LIN {X 0,Y 277.24,Z 414.573,A -85,B 0,C 180,E1 -17493.897,E2 -17493.897} C_VEL
LIN {X 0,Y 277.261,Z 414.56,A -85,B 0,C 180,E1 -17497.471,E2 -17497.471} C_VEL
LIN {X 0,Y 277.204,Z 414.578,A -85,B 0,C 180,E1 -17501.238,E2 -17501.238} C_VEL
LIN {X 0,Y 277.218,Z 414.568,A -85,B 0,C 180,E1 -17505.224,E2 -17505.224} C_VEL
LIN {X 0,Y 277.258,Z 414.57,A -85,B 0,C 180,E1 -17509.504,E2 -17509.504} C_VEL
LIN {X 0,Y 277.287,Z 414.57,A -85,B 0,C 180,E1 -17512.536,E2 -17512.536} C_VEL
LIN {X 0,Y 277.252,Z 414.575,A -85,B 0,C 180,E1 -17516.107,E2 -17516.107} C_VEL
LIN {X 0,Y 277.26,Z 414.568,A -85,B 0,C 180,E1 -17519.541,E2 -17519.541} C_VEL
LIN {X 0,Y 277.358,Z 414.56,A -85,B 0,C 180,E1 -17522.866,E2 -17522.866} C_VEL
LIN {X 0,Y 277.333,Z 414.568,A -85,B 0,C 180,E1 -17527.465,E2 -17527.465} C_VEL
LIN {X 0,Y 278.42,Z 417.605,A -85,B 0,C 180,E1 -17527.717,E2 -17527.717} C_VEL
LIN {X 0,Y 283.895,Z 430.25,A -85,B 0,C 180,E1 -17528.839,E2 -17528.839} C_VEL
LIN {X 0,Y 287.727,Z 441.564,A -85,B 0,C 180,E1 -17530.005,E2 -17530.005} C_VEL
LIN {X 0,Y 288.639,Z 445.273,A -85,B 0,C 180,E1 -17530.418,E2 -17530.418} C_VEL
LIN {X 0,Y 287.704,Z 456.27,A -85,B 0,C 180,E1 -17531.486,E2 -17531.486} C_VEL
LIN {X 0,Y 286.431,Z 467.423,A -85,B 0,C 180,E1 -17532.878,E2 -17532.878} C_VEL
LIN {X 0,Y 284.992,Z 477.37,A -85,B 0,C 180,E1 -17534.423,E2 -17534.423} C_VEL
LIN {X 0,Y 283.633,Z 485.752,A -85,B 0,C 180,E1 -17536.021,E2 -17536.021} C_VEL
LIN {X 0,Y 282.322,Z 493.35,A -85,B 0,C 180,E1 -17537.786,E2 -17537.786} C_VEL
LIN {X 0,Y 280.888,Z 500.786,A -85,B 0,C 180,E1 -17539.915,E2 -17539.915} C_VEL
LIN {X 0,Y 279.945,Z 506.702,A -85,B 0,C 180,E1 -17542.065,E2 -17542.065} C_VEL
LIN {X 0,Y 279.051,Z 511.413,A -85,B 0,C 180,E1 -17544.22,E2 -17544.22} C_VEL
LIN {X 0,Y 278.325,Z 515.036,A -85,B 0,C 180,E1 -17546.382,E2 -17546.382} C_VEL
LIN {X 0,Y 277.829,Z 517.669,A -85,B 0,C 180,E1 -17548.552,E2 -17548.552} C_VEL
LIN {X 0,Y 277.7,Z 519.747,A -85,B 0,C 180,E1 -17551.452,E2 -17551.452} C_VEL
LIN {X 0,Y 277.587,Z 520.2,A -85,B 0,C 180,E1 -17552.904,E2 -17552.904} C_VEL
LIN {X 0,Y 277.489,Z 520.279,A -85,B 0,C 180,E1 -17554.359,E2 -17554.359} C_VEL
LIN {X 0,Y 278.16,Z 519.232,A -85,B 0,C 180,E1 -17557.259,E2 -17557.259} C_VEL
LIN {X 0,Y 278.687,Z 518.077,A -85,B 0,C 180,E1 -17558.704,E2 -17558.704} C_VEL
LIN {X 0,Y 279.649,Z 514.63,A -85,B 0,C 180,E1 -17561.6,E2 -17561.6} C_VEL
LIN {X 0,Y 280.708,Z 510.847,A -85,B 0,C 180,E1 -17563.761,E2 -17563.761} C_VEL
LIN {X 0,Y 281.838,Z 505.952,A -85,B 0,C 180,E1 -17565.922,E2 -17565.922} C_VEL
LIN {X 0,Y 283.221,Z 499.731,A -85,B 0,C 180,E1 -17568.072,E2 -17568.072} C_VEL
LIN {X 0,Y 284.989,Z 491.93,A -85,B 0,C 180,E1 -17570.198,E2 -17570.198} C_VEL
LIN {X 0,Y 286.653,Z 483.93,A -85,B 0,C 180,E1 -17571.957,E2 -17571.957} C_VEL
LIN {X 0,Y 288.379,Z 474.102,A -85,B 0,C 180,E1 -17573.712,E2 -17573.712} C_VEL
LIN {X 0,Y 289.969,Z 462.99,A -85,B 0,C 180,E1 -17575.29,E2 -17575.29} C_VEL
LIN {X 0,Y 291.243,Z 452.011,A -85,B 0,C 180,E1 -17576.52,E2 -17576.52} C_VEL
LIN {X 0,Y 291.418,Z 448.805,A -85,B 0,C 180,E1 -17576.833,E2 -17576.833} C_VEL
LIN {X 0,Y 288.104,Z 438.67,A -85,B 0,C 180,E1 -17578.107,E2 -17578.107} C_VEL
LIN {X 0,Y 283.2,Z 426.913,A -85,B 0,C 180,E1 -17579.437,E2 -17579.437} C_VEL
LIN {X 0,Y 278.243,Z 417.384,A -85,B 0,C 180,E1 -17580.428,E2 -17580.428} C_VEL
LIN {X 0,Y 277.259,Z 414.575,A -85,B 0,C 180,E1 -17580.659,E2 -17580.659} C_VEL
LIN {X 0,Y 277.253,Z 414.579,A -85,B 0,C 180,E1 -17583.896,E2 -17583.896} C_VEL
LIN {X 0,Y 277.27,Z 414.557,A -85,B 0,C 180,E1 -17587.47,E2 -17587.47} C_VEL
LIN {X 0,Y 277.215,Z 414.579,A -85,B 0,C 180,E1 -17591.237,E2 -17591.237} C_VEL
LIN {X 0,Y 277.207,Z 414.574,A -85,B 0,C 180,E1 -17595.227,E2 -17595.227} C_VEL
LIN {X 0,Y 277.228,Z 414.555,A -85,B 0,C 180,E1 -17599.512,E2 -17599.512} C_VEL
LIN {X 0,Y 277.27,Z 414.542,A -85,B 0,C 180,E1 -17602.53,E2 -17602.53} C_VEL
LIN {X 0,Y 277.253,Z 414.573,A -85,B 0,C 180,E1 -17606.104,E2 -17606.104} C_VEL
LIN {X 0,Y 277.267,Z 414.524,A -85,B 0,C 180,E1 -17609.539,E2 -17609.539} C_VEL
LIN {X 0,Y 277.362,Z 414.537,A -85,B 0,C 180,E1 -17612.864,E2 -17612.864} C_VEL
LIN {X 0,Y 277.351,Z 414.616,A -85,B 0,C 180,E1 -17615.497,E2 -17615.497} C_VEL
LIN {X 0,Y 281.258,Z 428.661,A -85,B 0,C 180,E1 -17617.03,E2 -17617.03} C_VEL
LIN {X 0,Y 284.772,Z 441.274,A -85,B 0,C 180,E1 -17618.652,E2 -17618.652} C_VEL
LIN {X 0,Y 285.159,Z 442.879,A -85,B 0,C 180,E1 -17618.872,E2 -17618.872} C_VEL
LIN {X 0,Y 283.769,Z 455.996,A -85,B 0,C 180,E1 -17620.634,E2 -17620.634} C_VEL
LIN {X 0,Y 282.205,Z 468.131,A -85,B 0,C 180,E1 -17622.611,E2 -17622.611} C_VEL
LIN {X 0,Y 280.871,Z 479.118,A -85,B 0,C 180,E1 -17624.767,E2 -17624.767} C_VEL
LIN {X 0,Y 279.838,Z 488.37,A -85,B 0,C 180,E1 -17626.936,E2 -17626.936} C_VEL
LIN {X 0,Y 278.893,Z 497.005,A -85,B 0,C 180,E1 -17629.359,E2 -17629.359} C_VEL
LIN {X 0,Y 278.249,Z 504.77,A -85,B 0,C 180,E1 -17632.014,E2 -17632.014} C_VEL
LIN {X 0,Y 277.657,Z 509.994,A -85,B 0,C 180,E1 -17634.189,E2 -17634.189} C_VEL
LIN {X 0,Y 277.409,Z 514.29,A -85,B 0,C 180,E1 -17636.368,E2 -17636.368} C_VEL
LIN {X 0,Y 277.436,Z 515.059,A -85,B 0,C 180,E1 -17636.807,E2 -17636.807} C_VEL
LIN {X 0,Y 276.857,Z 517.048,A -85,B 0,C 180,E1 -17637.951,E2 -17637.951} C_VEL
LIN {X 0,Y 274.139,Z 520.047,A -85,B 0,C 180,E1 -17639.836,E2 -17639.836} C_VEL
LIN {X 0,Y 271.891,Z 522.007,A -85,B 0,C 180,E1 -17641.391,E2 -17641.391} C_VEL
LIN {X 0,Y 271.052,Z 523.132,A -85,B 0,C 180,E1 -17642.61,E2 -17642.61} C_VEL
LIN {X 0,Y 271.055,Z 523.425,A -85,B 0,C 180,E1 -17643.024,E2 -17643.024} C_VEL
LIN {X 0,Y 271.926,Z 525.003,A -85,B 0,C 180,E1 -17645.934,E2 -17645.934} C_VEL
LIN {X 0,Y 273.318,Z 525.329,A -85,B 0,C 180,E1 -17648.875,E2 -17648.875} C_VEL
LIN {X 0,Y 275.228,Z 524.402,A -85,B 0,C 180,E1 -17651.787,E2 -17651.787} C_VEL
LIN {X 0,Y 277.652,Z 522.226,A -85,B 0,C 180,E1 -17654.662,E2 -17654.662} C_VEL
LIN {X 0,Y 280.567,Z 518.782,A -85,B 0,C 180,E1 -17657.493,E2 -17657.493} C_VEL
LIN {X 0,Y 284.117,Z 513.978,A -85,B 0,C 180,E1 -17660.261,E2 -17660.261} C_VEL
LIN {X 0,Y 288.296,Z 507.671,A -85,B 0,C 180,E1 -17662.957,E2 -17662.957} C_VEL
LIN {X 0,Y 293.036,Z 499.73,A -85,B 0,C 180,E1 -17665.575,E2 -17665.575} C_VEL
LIN {X 0,Y 297.591,Z 491.324,A -85,B 0,C 180,E1 -17667.802,E2 -17667.802} C_VEL
LIN {X 0,Y 302.538,Z 481.329,A -85,B 0,C 180,E1 -17669.929,E2 -17669.929} C_VEL
LIN {X 0,Y 304.146,Z 477.942,A -85,B 0,C 180,E1 -17670.554,E2 -17670.554} C_VEL
LIN {X 0,Y 304.686,Z 476.205,A -85,B 0,C 180,E1 -17670.951,E2 -17670.951} C_VEL
LIN {X 0,Y 304.607,Z 471.254,A -85,B 0,C 180,E1 -17672.827,E2 -17672.827} C_VEL
LIN {X 0,Y 304.293,Z 469.306,A -85,B 0,C 180,E1 -17673.749,E2 -17673.749} C_VEL
LIN {X 0,Y 303.731,Z 468.086,A -85,B 0,C 180,E1 -17674.576,E2 -17674.576} C_VEL
LIN {X 0,Y 301.528,Z 465.974,A -85,B 0,C 180,E1 -17677.301,E2 -17677.301} C_VEL
LIN {X 0,Y 300.097,Z 465.624,A -85,B 0,C 180,E1 -17679.39,E2 -17679.39} C_VEL
LIN {X 0,Y 299.244,Z 466.047,A -85,B 0,C 180,E1 -17681.274,E2 -17681.274} C_VEL
LIN {X 0,Y 298.635,Z 467.442,A -85,B 0,C 180,E1 -17683.15,E2 -17683.15} C_VEL
LIN {X 0,Y 298.331,Z 471.007,A -85,B 0,C 180,E1 -17685.837,E2 -17685.837} C_VEL
LIN {X 0,Y 298.197,Z 472.343,A -85,B 0,C 180,E1 -17686.424,E2 -17686.424} C_VEL
LIN {X 0,Y 296.946,Z 480.691,A -85,B 0,C 180,E1 -17688.981,E2 -17688.981} C_VEL
LIN {X 0,Y 296.41,Z 486.651,A -85,B 0,C 180,E1 -17690.595,E2 -17690.595} C_VEL
LIN {X 0,Y 295.672,Z 495.118,A -85,B 0,C 180,E1 -17692.62,E2 -17692.62} C_VEL
LIN {X 0,Y 294.173,Z 507.873,A -85,B 0,C 180,E1 -17695.292,E2 -17695.292} C_VEL
LIN {X 0,Y 292.192,Z 518.62,A -85,B 0,C 180,E1 -17697.335,E2 -17697.335} C_VEL
LIN {X 0,Y 289.881,Z 527.876,A -85,B 0,C 180,E1 -17699.04,E2 -17699.04} C_VEL
LIN {X 0,Y 285.28,Z 541.73,A -85,B 0,C 180,E1 -17701.689,E2 -17701.689} C_VEL
LIN {X 0,Y 283.201,Z 548.047,A -85,B 0,C 180,E1 -17703.069,E2 -17703.069} C_VEL
LIN {X 0,Y 279.518,Z 556.829,A -85,B 0,C 180,E1 -17705.093,E2 -17705.093} C_VEL
LIN {X 0,Y 275.621,Z 566.892,A -85,B 0,C 180,E1 -17707.906,E2 -17707.906} C_VEL
LIN {X 0,Y 272.918,Z 574.417,A -85,B 0,C 180,E1 -17710.44,E2 -17710.44} C_VEL
LIN {X 0,Y 270.796,Z 581.627,A -85,B 0,C 180,E1 -17713.411,E2 -17713.411} C_VEL
LIN {X 0,Y 269.481,Z 587.459,A -85,B 0,C 180,E1 -17716.423,E2 -17716.423} C_VEL
LIN {X 0,Y 269.026,Z 591.968,A -85,B 0,C 180,E1 -17719.462,E2 -17719.462} C_VEL
LIN {X 0,Y 269.244,Z 595.321,A -85,B 0,C 180,E1 -17722.702,E2 -17722.702} C_VEL
LIN {X 0,Y 269.761,Z 597.078,A -85,B 0,C 180,E1 -17725.516,E2 -17725.516} C_VEL
LIN {X 0,Y 269.955,Z 597.987,A -85,B 0,C 180,E1 -17727.014,E2 -17727.014} C_VEL
LIN {X 0,Y 270.349,Z 598.479,A -85,B 0,C 180,E1 -17728.509,E2 -17728.509} C_VEL
LIN {X 0,Y 270.639,Z 598.546,A -85,B 0,C 180,E1 -17729.998,E2 -17729.998} C_VEL
LIN {X 0,Y 270.396,Z 598.125,A -85,B 0,C 180,E1 -17731.488,E2 -17731.488} C_VEL
LIN {X 0,Y 270.105,Z 597.237,A -85,B 0,C 180,E1 -17732.981,E2 -17732.981} C_VEL
LIN {X 0,Y 269.954,Z 595.925,A -85,B 0,C 180,E1 -17734.478,E2 -17734.478} C_VEL
LIN {X 0,Y 269.696,Z 593.115,A -85,B 0,C 180,E1 -17736.733,E2 -17736.733} C_VEL
LIN {X 0,Y 269.469,Z 589.213,A -85,B 0,C 180,E1 -17739.001,E2 -17739.001} C_VEL
LIN {X 0,Y 269.514,Z 584.144,A -85,B 0,C 180,E1 -17741.276,E2 -17741.276} C_VEL
LIN {X 0,Y 269.868,Z 577.764,A -85,B 0,C 180,E1 -17743.553,E2 -17743.553} C_VEL
LIN {X 0,Y 270.57,Z 570.514,A -85,B 0,C 180,E1 -17745.65,E2 -17745.65} C_VEL
LIN {X 0,Y 271.555,Z 561.767,A -85,B 0,C 180,E1 -17747.702,E2 -17747.702} C_VEL
LIN {X 0,Y 272.947,Z 551.946,A -85,B 0,C 180,E1 -17749.554,E2 -17749.554} C_VEL
LIN {X 0,Y 274.321,Z 541.032,A -85,B 0,C 180,E1 -17751.214,E2 -17751.214} C_VEL
LIN {X 0,Y 275.11,Z 532.003,A -85,B 0,C 180,E1 -17752.332,E2 -17752.332} C_VEL
LIN {X 0,Y 273.866,Z 512.707,A -85,B 0,C 180,E1 -17754.639,E2 -17754.639} C_VEL
LIN {X 0,Y 272.872,Z 498.445,A -85,B 0,C 180,E1 -17756.067,E2 -17756.067} C_VEL
LIN {X 0,Y 271.695,Z 482.747,A -85,B 0,C 180,E1 -17757.304,E2 -17757.304} C_VEL
LIN {X 0,Y 270.738,Z 469.018,A -85,B 0,C 180,E1 -17758.134,E2 -17758.134} C_VEL
LIN {X 0,Y 272.096,Z 458.724,A -85,B 0,C 180,E1 -17762.846,E2 -17762.846} C_VEL
LIN {X 0,Y 273.627,Z 449.25,A -85,B 0,C 180,E1 -17767.23,E2 -17767.23} C_VEL
LIN {X 0,Y 274.983,Z 441.851,A -85,B 0,C 180,E1 -17770.668,E2 -17770.668} C_VEL
LIN {X 0,Y 274.908,Z 438.792,A -85,B 0,C 180,E1 -17772.151,E2 -17772.151} C_VEL
LIN {X 0,Y 273.303,Z 431.108,A -85,B 0,C 180,E1 -17776.053,E2 -17776.053} C_VEL
LIN {X 0,Y 271.657,Z 422.876,A -85,B 0,C 180,E1 -17780.436,E2 -17780.436} C_VEL
LIN {X 0,Y 270.25,Z 415.448,A -85,B 0,C 180,E1 -17784.647,E2 -17784.647} C_VEL
LIN {X 0,Y 270.191,Z 415.455,A -85,B 0,C 180,E1 -17789.13,E2 -17789.13} C_VEL
LIN {X 0,Y 270.256,Z 415.444,A -85,B 0,C 180,E1 -17792.145,E2 -17792.145} C_VEL
LIN {X 0,Y 270.268,Z 415.443,A -85,B 0,C 180,E1 -17795.518,E2 -17795.518} C_VEL
LIN {X 0,Y 270.292,Z 415.435,A -85,B 0,C 180,E1 -17800.244,E2 -17800.244} C_VEL
LIN {X 0,Y 270.393,Z 415.425,A -85,B 0,C 180,E1 -17804.935,E2 -17804.935} C_VEL
LIN {X 0,Y 270.432,Z 415.417,A -85,B 0,C 180,E1 -17809.519,E2 -17809.519} C_VEL
LIN {X 0,Y 270.601,Z 415.402,A -85,B 0,C 180,E1 -17812.539,E2 -17812.539} C_VEL
LIN {X 0,Y 270.781,Z 415.38,A -85,B 0,C 180,E1 -17818.513,E2 -17818.513} C_VEL
LIN {X 0,Y 270.781,Z 415.377,A -85,B 0,C 180,E1 -17821.488,E2 -17821.488} C_VEL
LIN {X 0,Y 270.602,Z 415.388,A -85,B 0,C 180,E1 -17827.462,E2 -17827.462} C_VEL
LIN {X 0,Y 270.433,Z 415.408,A -85,B 0,C 180,E1 -17830.482,E2 -17830.482} C_VEL
LIN {X 0,Y 270.394,Z 415.428,A -85,B 0,C 180,E1 -17835.066,E2 -17835.066} C_VEL
LIN {X 0,Y 270.293,Z 415.439,A -85,B 0,C 180,E1 -17839.757,E2 -17839.757} C_VEL
LIN {X 0,Y 270.266,Z 415.445,A -85,B 0,C 180,E1 -17844.587,E2 -17844.587} C_VEL
LIN {X 0,Y 270.263,Z 415.437,A -85,B 0,C 180,E1 -17847.91,E2 -17847.91} C_VEL
LIN {X 0,Y 270.177,Z 415.447,A -85,B 0,C 180,E1 -17851.35,E2 -17851.35} C_VEL
LIN {X 0,Y 270.195,Z 415.451,A -85,B 0,C 180,E1 -17854.907,E2 -17854.907} C_VEL
LIN {X 0,Y 270.191,Z 415.441,A -85,B 0,C 180,E1 -17858.712,E2 -17858.712} C_VEL
LIN {X 0,Y 270.167,Z 415.453,A -85,B 0,C 180,E1 -17863.252,E2 -17863.252} C_VEL
LIN {X 0,Y 270.19,Z 415.452,A -85,B 0,C 180,E1 -17867.448,E2 -17867.448} C_VEL
LIN {X 0,Y 270.242,Z 415.442,A -85,B 0,C 180,E1 -17871.383,E2 -17871.383} C_VEL
LIN {X 0,Y 270.214,Z 415.45,A -85,B 0,C 180,E1 -17875.099,E2 -17875.099} C_VEL
LIN {X 0,Y 270.199,Z 415.447,A -85,B 0,C 180,E1 -17879.133,E2 -17879.133} C_VEL
LIN {X 0,Y 270.264,Z 415.442,A -85,B 0,C 180,E1 -17882.148,E2 -17882.148} C_VEL
LIN {X 0,Y 270.297,Z 415.444,A -85,B 0,C 180,E1 -17886.818,E2 -17886.818} C_VEL
LIN {X 0,Y 271.343,Z 418.376,A -85,B 0,C 180,E1 -17887.041,E2 -17887.041} C_VEL
LIN {X 0,Y 276.632,Z 430.499,A -85,B 0,C 180,E1 -17888.154,E2 -17888.154} C_VEL
LIN {X 0,Y 280.118,Z 439.972,A -85,B 0,C 180,E1 -17889.162,E2 -17889.162} C_VEL
LIN {X 0,Y 282.052,Z 446.798,A -85,B 0,C 180,E1 -17889.944,E2 -17889.944} C_VEL
LIN {X 0,Y 281.102,Z 457.619,A -85,B 0,C 180,E1 -17891.035,E2 -17891.035} C_VEL
LIN {X 0,Y 279.754,Z 468.707,A -85,B 0,C 180,E1 -17892.456,E2 -17892.456} C_VEL
LIN {X 0,Y 278.239,Z 478.779,A -85,B 0,C 180,E1 -17894.066,E2 -17894.066} C_VEL
LIN {X 0,Y 276.844,Z 486.952,A -85,B 0,C 180,E1 -17895.671,E2 -17895.671} C_VEL
LIN {X 0,Y 275.476,Z 494.519,A -85,B 0,C 180,E1 -17897.477,E2 -17897.477} C_VEL
LIN {X 0,Y 273.988,Z 501.915,A -85,B 0,C 180,E1 -17899.658,E2 -17899.658} C_VEL
LIN {X 0,Y 273.008,Z 507.806,A -85,B 0,C 180,E1 -17901.862,E2 -17901.862} C_VEL
LIN {X 0,Y 272.07,Z 512.497,A -85,B 0,C 180,E1 -17904.071,E2 -17904.071} C_VEL
LIN {X 0,Y 271.316,Z 516.101,A -85,B 0,C 180,E1 -17906.289,E2 -17906.289} C_VEL
LIN {X 0,Y 270.807,Z 518.715,A -85,B 0,C 180,E1 -17908.515,E2 -17908.515} C_VEL
LIN {X 0,Y 270.676,Z 520.77,A -85,B 0,C 180,E1 -17911.489,E2 -17911.489} C_VEL
LIN {X 0,Y 270.565,Z 521.209,A -85,B 0,C 180,E1 -17912.979,E2 -17912.979} C_VEL
LIN {X 0,Y 270.474,Z 521.279,A -85,B 0,C 180,E1 -17914.472,E2 -17914.472} C_VEL
LIN {X 0,Y 271.186,Z 520.206,A -85,B 0,C 180,E1 -17917.447,E2 -17917.447} C_VEL
LIN {X 0,Y 271.738,Z 519.038,A -85,B 0,C 180,E1 -17918.929,E2 -17918.929} C_VEL
LIN {X 0,Y 272.614,Z 516.012,A -85,B 0,C 180,E1 -17921.578,E2 -17921.578} C_VEL
LIN {X 0,Y 273.87,Z 511.766,A -85,B 0,C 180,E1 -17924.112,E2 -17924.112} C_VEL
LIN {X 0,Y 275.072,Z 506.841,A -85,B 0,C 180,E1 -17926.324,E2 -17926.324} C_VEL
LIN {X 0,Y 276.531,Z 500.591,A -85,B 0,C 180,E1 -17928.525,E2 -17928.525} C_VEL
LIN {X 0,Y 278.383,Z 492.759,A -85,B 0,C 180,E1 -17930.699,E2 -17930.699} C_VEL
LIN {X 0,Y 280.109,Z 484.724,A -85,B 0,C 180,E1 -17932.498,E2 -17932.498} C_VEL
LIN {X 0,Y 281.922,Z 474.827,A -85,B 0,C 180,E1 -17934.29,E2 -17934.29} C_VEL
LIN {X 0,Y 283.598,Z 463.653,A -85,B 0,C 180,E1 -17935.9,E2 -17935.9} C_VEL
LIN {X 0,Y 284.932,Z 452.571,A -85,B 0,C 180,E1 -17937.155,E2 -17937.155} C_VEL
LIN {X 0,Y 284.907,Z 450.551,A -85,B 0,C 180,E1 -17937.371,E2 -17937.371} C_VEL
LIN {X 0,Y 281.543,Z 440.304,A -85,B 0,C 180,E1 -17938.72,E2 -17938.72} C_VEL
LIN {X 0,Y 276.669,Z 428.718,A -85,B 0,C 180,E1 -17940.106,E2 -17940.106} C_VEL
LIN {X 0,Y 270.532,Z 416.857,A -85,B 0,C 180,E1 -17941.381,E2 -17941.381} C_VEL
LIN {X 0,Y 270.215,Z 415.455,A -85,B 0,C 180,E1 -17941.509,E2 -17941.509} C_VEL
LIN {X 0,Y 270.208,Z 415.453,A -85,B 0,C 180,E1 -17944.906,E2 -17944.906} C_VEL
LIN {X 0,Y 270.203,Z 415.434,A -85,B 0,C 180,E1 -17948.711,E2 -17948.711} C_VEL
LIN {X 0,Y 270.177,Z 415.451,A -85,B 0,C 180,E1 -17952.559,E2 -17952.559} C_VEL
LIN {X 0,Y 270.171,Z 415.455,A -85,B 0,C 180,E1 -17956.751,E2 -17956.751} C_VEL
LIN {X 0,Y 270.18,Z 415.433,A -85,B 0,C 180,E1 -17959.435,E2 -17959.435} C_VEL
LIN {X 0,Y 270.231,Z 415.439,A -85,B 0,C 180,E1 -17963.731,E2 -17963.731} C_VEL
LIN {X 0,Y 270.209,Z 415.446,A -85,B 0,C 180,E1 -17966.893,E2 -17966.893} C_VEL
LIN {X 0,Y 270.201,Z 415.4,A -85,B 0,C 180,E1 -17970.383,E2 -17970.383} C_VEL
LIN {X 0,Y 270.271,Z 415.432,A -85,B 0,C 180,E1 -17973.764,E2 -17973.764} C_VEL
LIN {X 0,Y 270.302,Z 415.439,A -85,B 0,C 180,E1 -17975.14,E2 -17975.14} C_VEL
LIN {X 0,Y 274.353,Z 430.011,A -85,B 0,C 180,E1 -17976.782,E2 -17976.782} C_VEL
LIN {X 0,Y 277.882,Z 442.84,A -85,B 0,C 180,E1 -17978.486,E2 -17978.486} C_VEL
LIN {X 0,Y 277.989,Z 445.861,A -85,B 0,C 180,E1 -17978.883,E2 -17978.883} C_VEL
LIN {X 0,Y 276.524,Z 458.707,A -85,B 0,C 180,E1 -17980.706,E2 -17980.706} C_VEL
LIN {X 0,Y 274.853,Z 471.464,A -85,B 0,C 180,E1 -17982.899,E2 -17982.899} C_VEL
LIN {X 0,Y 273.639,Z 482.105,A -85,B 0,C 180,E1 -17985.117,E2 -17985.117} C_VEL
LIN {X 0,Y 272.548,Z 491.055,A -85,B 0,C 180,E1 -17987.338,E2 -17987.338} C_VEL
LIN {X 0,Y 271.627,Z 499.757,A -85,B 0,C 180,E1 -17989.941,E2 -17989.941} C_VEL
LIN {X 0,Y 271.015,Z 506.913,A -85,B 0,C 180,E1 -17992.55,E2 -17992.55} C_VEL
LIN {X 0,Y 270.323,Z 513.495,A -85,B 0,C 180,E1 -17995.526,E2 -17995.526} C_VEL
LIN {X 0,Y 270.608,Z 518.481,A -85,B 0,C 180,E1 -17998.511,E2 -17998.511} C_VEL
LIN {X 0,Y 270.775,Z 522.096,A -85,B 0,C 180,E1 -18001.487,E2 -18001.487} C_VEL
LIN {X 0,Y 271.055,Z 523.425,A -85,B 0,C 180,E1 -18003.024,E2 -18003.024} C_VEL
LIN {X 0,Y 270.711,Z 524.355,A -85,B 0,C 180,E1 -18004.258,E2 -18004.258} C_VEL
LIN {X 0,Y 268.585,Z 525.695,A -85,B 0,C 180,E1 -18006.295,E2 -18006.295} C_VEL
LIN {X 0,Y 266.947,Z 526.486,A -85,B 0,C 180,E1 -18007.95,E2 -18007.95} C_VEL
LIN {X 0,Y 266.608,Z 526.719,A -85,B 0,C 180,E1 -18009.217,E2 -18009.217} C_VEL
LIN {X 0,Y 266.778,Z 526.675,A -85,B 0,C 180,E1 -18009.639,E2 -18009.639} C_VEL
LIN {X 0,Y 268.492,Z 526.036,A -85,B 0,C 180,E1 -18012.087,E2 -18012.087} C_VEL
LIN {X 0,Y 271.04,Z 524.091,A -85,B 0,C 180,E1 -18015.028,E2 -18015.028} C_VEL
LIN {X 0,Y 274.111,Z 520.899,A -85,B 0,C 180,E1 -18017.919,E2 -18017.919} C_VEL
LIN {X 0,Y 277.856,Z 516.368,A -85,B 0,C 180,E1 -18020.739,E2 -18020.739} C_VEL
LIN {X 0,Y 282.257,Z 510.418,A -85,B 0,C 180,E1 -18023.477,E2 -18023.477} C_VEL
LIN {X 0,Y 287.225,Z 502.921,A -85,B 0,C 180,E1 -18026.131,E2 -18026.131} C_VEL
LIN {X 0,Y 292.722,Z 493.658,A -85,B 0,C 180,E1 -18028.697,E2 -18028.697} C_VEL
LIN {X 0,Y 297.977,Z 483.982,A -85,B 0,C 180,E1 -18030.835,E2 -18030.835} C_VEL
LIN {X 0,Y 299.576,Z 480.808,A -85,B 0,C 180,E1 -18031.441,E2 -18031.441} C_VEL
LIN {X 0,Y 299.948,Z 477.648,A -85,B 0,C 180,E1 -18032.609,E2 -18032.609} C_VEL
LIN {X 0,Y 299.973,Z 475.862,A -85,B 0,C 180,E1 -18033.4,E2 -18033.4} C_VEL
LIN {X 0,Y 299.435,Z 473.689,A -85,B 0,C 180,E1 -18034.765,E2 -18034.765} C_VEL
LIN {X 0,Y 298.013,Z 472.253,A -85,B 0,C 180,E1 -18036.694,E2 -18036.694} C_VEL
LIN {X 0,Y 296.786,Z 471.701,A -85,B 0,C 180,E1 -18038.605,E2 -18038.605} C_VEL
LIN {X 0,Y 295.829,Z 471.944,A -85,B 0,C 180,E1 -18040.515,E2 -18040.515} C_VEL
LIN {X 0,Y 295.192,Z 473.041,A -85,B 0,C 180,E1 -18042.432,E2 -18042.432} C_VEL
LIN {X 0,Y 294.724,Z 475.151,A -85,B 0,C 180,E1 -18044.324,E2 -18044.324} C_VEL
LIN {X 0,Y 294.537,Z 477.31,A -85,B 0,C 180,E1 -18045.711,E2 -18045.711} C_VEL
LIN {X 0,Y 293.044,Z 484.352,A -85,B 0,C 180,E1 -18048.027,E2 -18048.027} C_VEL
LIN {X 0,Y 291.904,Z 491.714,A -85,B 0,C 180,E1 -18050.106,E2 -18050.106} C_VEL
LIN {X 0,Y 290.914,Z 498.87,A -85,B 0,C 180,E1 -18051.901,E2 -18051.901} C_VEL
LIN {X 0,Y 289.088,Z 509.654,A -85,B 0,C 180,E1 -18054.304,E2 -18054.304} C_VEL
LIN {X 0,Y 286.905,Z 519.89,A -85,B 0,C 180,E1 -18056.394,E2 -18056.394} C_VEL
LIN {X 0,Y 284.111,Z 529.513,A -85,B 0,C 180,E1 -18058.286,E2 -18058.286} C_VEL
LIN {X 0,Y 279.143,Z 542.919,A -85,B 0,C 180,E1 -18061.008,E2 -18061.008} C_VEL
LIN {X 0,Y 276.306,Z 550.428,A -85,B 0,C 180,E1 -18062.751,E2 -18062.751} C_VEL
LIN {X 0,Y 272.536,Z 558.765,A -85,B 0,C 180,E1 -18064.853,E2 -18064.853} C_VEL
LIN {X 0,Y 268.572,Z 568.137,A -85,B 0,C 180,E1 -18067.7,E2 -18067.7} C_VEL
LIN {X 0,Y 265.514,Z 576.106,A -85,B 0,C 180,E1 -18070.677,E2 -18070.677} C_VEL
LIN {X 0,Y 263.407,Z 582.915,A -85,B 0,C 180,E1 -18073.846,E2 -18073.846} C_VEL
LIN {X 0,Y 262.287,Z 587.984,A -85,B 0,C 180,E1 -18076.833,E2 -18076.833} C_VEL
LIN {X 0,Y 261.954,Z 591.075,A -85,B 0,C 180,E1 -18079.174,E2 -18079.174} C_VEL
LIN {X 0,Y 262.181,Z 594.385,A -85,B 0,C 180,E1 -18082.665,E2 -18082.665} C_VEL
LIN {X 0,Y 262.71,Z 596.092,A -85,B 0,C 180,E1 -18085.395,E2 -18085.395} C_VEL
LIN {X 0,Y 262.894,Z 596.987,A -85,B 0,C 180,E1 -18086.934,E2 -18086.934} C_VEL
LIN {X 0,Y 263.304,Z 597.475,A -85,B 0,C 180,E1 -18088.469,E2 -18088.469} C_VEL
LIN {X 0,Y 263.608,Z 597.537,A -85,B 0,C 180,E1 -18089.998,E2 -18089.998} C_VEL
LIN {X 0,Y 263.357,Z 597.107,A -85,B 0,C 180,E1 -18091.528,E2 -18091.528} C_VEL
LIN {X 0,Y 263.047,Z 596.201,A -85,B 0,C 180,E1 -18093.061,E2 -18093.061} C_VEL
LIN {X 0,Y 262.902,Z 594.881,A -85,B 0,C 180,E1 -18094.598,E2 -18094.598} C_VEL
LIN {X 0,Y 262.615,Z 592.047,A -85,B 0,C 180,E1 -18096.915,E2 -18096.915} C_VEL
LIN {X 0,Y 262.381,Z 588.122,A -85,B 0,C 180,E1 -18099.246,E2 -18099.246} C_VEL
LIN {X 0,Y 262.442,Z 583.029,A -85,B 0,C 180,E1 -18101.584,E2 -18101.584} C_VEL
LIN {X 0,Y 262.876,Z 576.634,A -85,B 0,C 180,E1 -18103.921,E2 -18103.921} C_VEL
LIN {X 0,Y 263.665,Z 569.005,A -85,B 0,C 180,E1 -18106.168,E2 -18106.168} C_VEL
LIN {X 0,Y 264.703,Z 560.575,A -85,B 0,C 180,E1 -18108.176,E2 -18108.176} C_VEL
LIN {X 0,Y 266.167,Z 550.721,A -85,B 0,C 180,E1 -18110.074,E2 -18110.074} C_VEL
LIN {X 0,Y 267.458,Z 541.078,A -85,B 0,C 180,E1 -18111.583,E2 -18111.583} C_VEL
LIN {X 0,Y 268.208,Z 532.27,A -85,B 0,C 180,E1 -18112.735,E2 -18112.735} C_VEL
LIN {X 0,Y 267.392,Z 520.106,A -85,B 0,C 180,E1 -18114.142,E2 -18114.142} C_VEL
LIN {X 0,Y 266.398,Z 507.297,A -85,B 0,C 180,E1 -18115.43,E2 -18115.43} C_VEL
LIN {X 0,Y 265.388,Z 492.373,A -85,B 0,C 180,E1 -18116.86,E2 -18116.86} C_VEL
LIN {X 0,Y 264.268,Z 476.728,A -85,B 0,C 180,E1 -18118.03,E2 -18118.03} C_VEL
LIN {X 0,Y 263.744,Z 468.058,A -85,B 0,C 180,E1 -18118.565,E2 -18118.565} C_VEL
LIN {X 0,Y 265.007,Z 458.825,A -85,B 0,C 180,E1 -18122.931,E2 -18122.931} C_VEL
LIN {X 0,Y 266.574,Z 449.575,A -85,B 0,C 180,E1 -18127.325,E2 -18127.325} C_VEL
LIN {X 0,Y 267.95,Z 442.012,A -85,B 0,C 180,E1 -18130.971,E2 -18130.971} C_VEL
LIN {X 0,Y 267.646,Z 438.607,A -85,B 0,C 180,E1 -18132.673,E2 -18132.673} C_VEL
LIN {X 0,Y 265.816,Z 429.824,A -85,B 0,C 180,E1 -18137.294,E2 -18137.294} C_VEL
LIN {X 0,Y 264.351,Z 422.504,A -85,B 0,C 180,E1 -18141.335,E2 -18141.335} C_VEL
LIN {X 0,Y 263.174,Z 416.33,A -85,B 0,C 180,E1 -18144.961,E2 -18144.961} C_VEL
LIN {X 0,Y 263.142,Z 416.33,A -85,B 0,C 180,E1 -18149.506,E2 -18149.506} C_VEL
LIN {X 0,Y 263.186,Z 416.328,A -85,B 0,C 180,E1 -18153.002,E2 -18153.002} C_VEL
LIN {X 0,Y 263.175,Z 416.325,A -85,B 0,C 180,E1 -18156.386,E2 -18156.386} C_VEL
LIN {X 0,Y 263.254,Z 416.312,A -85,B 0,C 180,E1 -18159.693,E2 -18159.693} C_VEL
LIN {X 0,Y 263.341,Z 416.304,A -85,B 0,C 180,E1 -18164.522,E2 -18164.522} C_VEL
LIN {X 0,Y 263.365,Z 416.299,A -85,B 0,C 180,E1 -18169.234,E2 -18169.234} C_VEL
LIN {X 0,Y 263.563,Z 416.278,A -85,B 0,C 180,E1 -18172.338,E2 -18172.338} C_VEL
LIN {X 0,Y 263.745,Z 416.257,A -85,B 0,C 180,E1 -18178.473,E2 -18178.473} C_VEL
LIN {X 0,Y 263.746,Z 416.254,A -85,B 0,C 180,E1 -18181.527,E2 -18181.527} C_VEL
LIN {X 0,Y 263.563,Z 416.263,A -85,B 0,C 180,E1 -18187.662,E2 -18187.662} C_VEL
LIN {X 0,Y 263.365,Z 416.29,A -85,B 0,C 180,E1 -18190.766,E2 -18190.766} C_VEL
LIN {X 0,Y 263.342,Z 416.304,A -85,B 0,C 180,E1 -18195.479,E2 -18195.479} C_VEL
LIN {X 0,Y 263.255,Z 416.318,A -85,B 0,C 180,E1 -18200.308,E2 -18200.308} C_VEL
LIN {X 0,Y 263.201,Z 416.323,A -85,B 0,C 180,E1 -18205.293,E2 -18205.293} C_VEL
LIN {X 0,Y 263.159,Z 416.311,A -85,B 0,C 180,E1 -18208.733,E2 -18208.733} C_VEL
LIN {X 0,Y 263.126,Z 416.327,A -85,B 0,C 180,E1 -18212.29,E2 -18212.29} C_VEL
LIN {X 0,Y 263.176,Z 416.317,A -85,B 0,C 180,E1 -18216.765,E2 -18216.765} C_VEL
LIN {X 0,Y 263.12,Z 416.333,A -85,B 0,C 180,E1 -18221.596,E2 -18221.596} C_VEL
LIN {X 0,Y 263.129,Z 416.323,A -85,B 0,C 180,E1 -18226.02,E2 -18226.02} C_VEL
LIN {X 0,Y 263.136,Z 416.328,A -85,B 0,C 180,E1 -18230.136,E2 -18230.136} C_VEL
LIN {X 0,Y 263.188,Z 416.327,A -85,B 0,C 180,E1 -18234.025,E2 -18234.025} C_VEL
LIN {X 0,Y 263.132,Z 416.332,A -85,B 0,C 180,E1 -18237.714,E2 -18237.714} C_VEL
LIN {X 0,Y 263.2,Z 416.323,A -85,B 0,C 180,E1 -18241.785,E2 -18241.785} C_VEL
LIN {X 0,Y 263.26,Z 416.321,A -85,B 0,C 180,E1 -18246.093,E2 -18246.093} C_VEL
LIN {X 0,Y 264.369,Z 419.315,A -85,B 0,C 180,E1 -18246.343,E2 -18246.343} C_VEL
LIN {X 0,Y 269.901,Z 431.846,A -85,B 0,C 180,E1 -18247.551,E2 -18247.551} C_VEL
LIN {X 0,Y 273.537,Z 441.717,A -85,B 0,C 180,E1 -18248.652,E2 -18248.652} C_VEL
LIN {X 0,Y 275.451,Z 448.337,A -85,B 0,C 180,E1 -18249.449,E2 -18249.449} C_VEL
LIN {X 0,Y 274.317,Z 460.469,A -85,B 0,C 180,E1 -18250.742,E2 -18250.742} C_VEL
LIN {X 0,Y 272.922,Z 471.272,A -85,B 0,C 180,E1 -18252.204,E2 -18252.204} C_VEL
LIN {X 0,Y 271.367,Z 480.983,A -85,B 0,C 180,E1 -18253.839,E2 -18253.839} C_VEL
LIN {X 0,Y 269.717,Z 489.765,A -85,B 0,C 180,E1 -18255.67,E2 -18255.67} C_VEL
LIN {X 0,Y 268.111,Z 498.303,A -85,B 0,C 180,E1 -18257.897,E2 -18257.897} C_VEL
LIN {X 0,Y 266.689,Z 505.178,A -85,B 0,C 180,E1 -18260.139,E2 -18260.139} C_VEL
LIN {X 0,Y 265.754,Z 510.608,A -85,B 0,C 180,E1 -18262.403,E2 -18262.403} C_VEL
LIN {X 0,Y 264.817,Z 514.902,A -85,B 0,C 180,E1 -18264.672,E2 -18264.672} C_VEL
LIN {X 0,Y 264.067,Z 518.156,A -85,B 0,C 180,E1 -18266.95,E2 -18266.95} C_VEL
LIN {X 0,Y 263.666,Z 520.97,A -85,B 0,C 180,E1 -18270.002,E2 -18270.002} C_VEL
LIN {X 0,Y 263.652,Z 521.792,A -85,B 0,C 180,E1 -18271.529,E2 -18271.529} C_VEL
LIN {X 0,Y 263.46,Z 522.28,A -85,B 0,C 180,E1 -18274.592,E2 -18274.592} C_VEL
LIN {X 0,Y 263.743,Z 521.933,A -85,B 0,C 180,E1 -18276.12,E2 -18276.12} C_VEL
LIN {X 0,Y 264.216,Z 521.179,A -85,B 0,C 180,E1 -18277.644,E2 -18277.644} C_VEL
LIN {X 0,Y 264.794,Z 520,A -85,B 0,C 180,E1 -18279.165,E2 -18279.165} C_VEL
LIN {X 0,Y 265.716,Z 516.978,A -85,B 0,C 180,E1 -18281.865,E2 -18281.865} C_VEL
LIN {X 0,Y 267.02,Z 512.687,A -85,B 0,C 180,E1 -18284.481,E2 -18284.481} C_VEL
LIN {X 0,Y 268.32,Z 507.728,A -85,B 0,C 180,E1 -18286.747,E2 -18286.747} C_VEL
LIN {X 0,Y 269.859,Z 501.451,A -85,B 0,C 180,E1 -18289,E2 -18289} C_VEL
LIN {X 0,Y 271.793,Z 493.59,A -85,B 0,C 180,E1 -18291.225,E2 -18291.225} C_VEL
LIN {X 0,Y 273.609,Z 485.518,A -85,B 0,C 180,E1 -18293.063,E2 -18293.063} C_VEL
LIN {X 0,Y 275.503,Z 475.555,A -85,B 0,C 180,E1 -18294.893,E2 -18294.893} C_VEL
LIN {X 0,Y 277.266,Z 464.319,A -85,B 0,C 180,E1 -18296.537,E2 -18296.537} C_VEL
LIN {X 0,Y 278.504,Z 454.259,A -85,B 0,C 180,E1 -18297.705,E2 -18297.705} C_VEL
LIN {X 0,Y 278.413,Z 452.345,A -85,B 0,C 180,E1 -18297.93,E2 -18297.93} C_VEL
LIN {X 0,Y 275.148,Z 442.353,A -85,B 0,C 180,E1 -18299.312,E2 -18299.312} C_VEL
LIN {X 0,Y 270.337,Z 430.971,A -85,B 0,C 180,E1 -18300.754,E2 -18300.754} C_VEL
LIN {X 0,Y 264.424,Z 419.548,A -85,B 0,C 180,E1 -18302.078,E2 -18302.078} C_VEL
LIN {X 0,Y 263.243,Z 416.859,A -85,B 0,C 180,E1 -18302.325,E2 -18302.325} C_VEL
LIN {X 0,Y 263.184,Z 416.329,A -85,B 0,C 180,E1 -18302.368,E2 -18302.368} C_VEL
LIN {X 0,Y 263.187,Z 416.318,A -85,B 0,C 180,E1 -18306.764,E2 -18306.764} C_VEL
LIN {X 0,Y 263.13,Z 416.332,A -85,B 0,C 180,E1 -18311.594,E2 -18311.594} C_VEL
LIN {X 0,Y 263.129,Z 416.334,A -85,B 0,C 180,E1 -18313.985,E2 -18313.985} C_VEL
LIN {X 0,Y 263.13,Z 416.328,A -85,B 0,C 180,E1 -18318.407,E2 -18318.407} C_VEL
LIN {X 0,Y 263.165,Z 416.293,A -85,B 0,C 180,E1 -18322.103,E2 -18322.103} C_VEL
LIN {X 0,Y 263.157,Z 416.331,A -85,B 0,C 180,E1 -18325.886,E2 -18325.886} C_VEL
LIN {X 0,Y 263.146,Z 416.281,A -85,B 0,C 180,E1 -18329.506,E2 -18329.506} C_VEL
LIN {X 0,Y 263.199,Z 416.302,A -85,B 0,C 180,E1 -18333.003,E2 -18333.003} C_VEL
LIN {X 0,Y 263.297,Z 416.499,A -85,B 0,C 180,E1 -18334.818,E2 -18334.818} C_VEL
LIN {X 0,Y 267.184,Z 430.795,A -85,B 0,C 180,E1 -18336.462,E2 -18336.462} C_VEL
LIN {X 0,Y 270.567,Z 442.838,A -85,B 0,C 180,E1 -18338.094,E2 -18338.094} C_VEL
LIN {X 0,Y 271.096,Z 445.914,A -85,B 0,C 180,E1 -18338.526,E2 -18338.526} C_VEL
LIN {X 0,Y 269.611,Z 458.866,A -85,B 0,C 180,E1 -18340.39,E2 -18340.39} C_VEL
LIN {X 0,Y 268.03,Z 470.768,A -85,B 0,C 180,E1 -18342.449,E2 -18342.449} C_VEL
LIN {X 0,Y 266.694,Z 481.668,A -85,B 0,C 180,E1 -18344.72,E2 -18344.72} C_VEL
LIN {X 0,Y 265.577,Z 490.848,A -85,B 0,C 180,E1 -18347,E2 -18347} C_VEL
LIN {X 0,Y 264.646,Z 499.629,A -85,B 0,C 180,E1 -18349.606,E2 -18349.606} C_VEL
LIN {X 0,Y 263.974,Z 507.204,A -85,B 0,C 180,E1 -18352.35,E2 -18352.35} C_VEL
LIN {X 0,Y 263.274,Z 513.964,A -85,B 0,C 180,E1 -18355.406,E2 -18355.406} C_VEL
LIN {X 0,Y 263.56,Z 519.14,A -85,B 0,C 180,E1 -18358.472,E2 -18358.472} C_VEL
LIN {X 0,Y 263.753,Z 522.955,A -85,B 0,C 180,E1 -18361.527,E2 -18361.527} C_VEL
LIN {X 0,Y 264.448,Z 525.439,A -85,B 0,C 180,E1 -18364.573,E2 -18364.573} C_VEL
LIN {X 0,Y 265.66,Z 526.63,A -85,B 0,C 180,E1 -18367.601,E2 -18367.601} C_VEL
LIN {X 0,Y 266.778,Z 526.675,A -85,B 0,C 180,E1 -18369.639,E2 -18369.639} C_VEL
LIN {X 0,Y 266.956,Z 526.602,A -85,B 0,C 180,E1 -18370.907,E2 -18370.907} C_VEL
LIN {X 0,Y 265.754,Z 526.478,A -85,B 0,C 180,E1 -18373.025,E2 -18373.025} C_VEL
LIN {X 0,Y 264.881,Z 526.092,A -85,B 0,C 180,E1 -18374.728,E2 -18374.728} C_VEL
LIN {X 0,Y 265.104,Z 525.433,A -85,B 0,C 180,E1 -18375.996,E2 -18375.996} C_VEL
LIN {X 0,Y 265.454,Z 525.079,A -85,B 0,C 180,E1 -18376.409,E2 -18376.409} C_VEL
LIN {X 0,Y 267.702,Z 523.04,A -85,B 0,C 180,E1 -18378.363,E2 -18378.363} C_VEL
LIN {X 0,Y 271.649,Z 518.8,A -85,B 0,C 180,E1 -18381.235,E2 -18381.235} C_VEL
LIN {X 0,Y 276.243,Z 513.175,A -85,B 0,C 180,E1 -18384.02,E2 -18384.02} C_VEL
LIN {X 0,Y 282.151,Z 505.12,A -85,B 0,C 180,E1 -18387.038,E2 -18387.038} C_VEL
LIN {X 0,Y 287.96,Z 496.121,A -85,B 0,C 180,E1 -18389.618,E2 -18389.618} C_VEL
LIN {X 0,Y 293.593,Z 486.648,A -85,B 0,C 180,E1 -18391.778,E2 -18391.778} C_VEL
LIN {X 0,Y 294.528,Z 484.979,A -85,B 0,C 180,E1 -18392.11,E2 -18392.11} C_VEL
LIN {X 0,Y 295.014,Z 483.647,A -85,B 0,C 180,E1 -18392.496,E2 -18392.496} C_VEL
LIN {X 0,Y 295.286,Z 481.232,A -85,B 0,C 180,E1 -18393.588,E2 -18393.588} C_VEL
LIN {X 0,Y 295.071,Z 479.26,A -85,B 0,C 180,E1 -18394.864,E2 -18394.864} C_VEL
LIN {X 0,Y 293.9,Z 478.017,A -85,B 0,C 180,E1 -18396.714,E2 -18396.714} C_VEL
LIN {X 0,Y 292.807,Z 477.607,A -85,B 0,C 180,E1 -18398.613,E2 -18398.613} C_VEL
LIN {X 0,Y 291.94,Z 477.951,A -85,B 0,C 180,E1 -18400.54,E2 -18400.54} C_VEL
LIN {X 0,Y 291.302,Z 479.221,A -85,B 0,C 180,E1 -18402.495,E2 -18402.495} C_VEL
LIN {X 0,Y 290.814,Z 481.557,A -85,B 0,C 180,E1 -18404.494,E2 -18404.494} C_VEL
LIN {X 0,Y 290.44,Z 483.363,A -85,B 0,C 180,E1 -18405.432,E2 -18405.432} C_VEL
LIN {X 0,Y 288.76,Z 489.539,A -85,B 0,C 180,E1 -18407.518,E2 -18407.518} C_VEL
LIN {X 0,Y 287.224,Z 496.921,A -85,B 0,C 180,E1 -18409.692,E2 -18409.692} C_VEL
LIN {X 0,Y 285.655,Z 504.68,A -85,B 0,C 180,E1 -18411.685,E2 -18411.685} C_VEL
LIN {X 0,Y 283.497,Z 514.341,A -85,B 0,C 180,E1 -18413.929,E2 -18413.929} C_VEL
LIN {X 0,Y 280.734,Z 524.377,A -85,B 0,C 180,E1 -18416.078,E2 -18416.078} C_VEL
LIN {X 0,Y 277.006,Z 534.705,A -85,B 0,C 180,E1 -18418.232,E2 -18418.232} C_VEL
LIN {X 0,Y 271.953,Z 547.052,A -85,B 0,C 180,E1 -18421.016,E2 -18421.016} C_VEL
LIN {X 0,Y 267.972,Z 555.271,A -85,B 0,C 180,E1 -18423.088,E2 -18423.088} C_VEL
LIN {X 0,Y 263.489,Z 564.96,A -85,B 0,C 180,E1 -18425.997,E2 -18425.997} C_VEL
LIN {X 0,Y 260.192,Z 572.183,A -85,B 0,C 180,E1 -18428.613,E2 -18428.613} C_VEL
LIN {X 0,Y 257.571,Z 579.166,A -85,B 0,C 180,E1 -18431.711,E2 -18431.711} C_VEL
LIN {X 0,Y 255.812,Z 584.845,A -85,B 0,C 180,E1 -18434.869,E2 -18434.869} C_VEL
LIN {X 0,Y 255.096,Z 588.307,A -85,B 0,C 180,E1 -18437.266,E2 -18437.266} C_VEL
LIN {X 0,Y 254.877,Z 591.783,A -85,B 0,C 180,E1 -18440.475,E2 -18440.475} C_VEL
LIN {X 0,Y 255.639,Z 595.102,A -85,B 0,C 180,E1 -18445.267,E2 -18445.267} C_VEL
LIN {X 0,Y 255.833,Z 595.987,A -85,B 0,C 180,E1 -18446.849,E2 -18446.849} C_VEL
LIN {X 0,Y 256.26,Z 596.472,A -85,B 0,C 180,E1 -18448.427,E2 -18448.427} C_VEL
LIN {X 0,Y 256.577,Z 596.529,A -85,B 0,C 180,E1 -18449.998,E2 -18449.998} C_VEL
LIN {X 0,Y 256.317,Z 596.087,A -85,B 0,C 180,E1 -18451.569,E2 -18451.569} C_VEL
LIN {X 0,Y 255.99,Z 595.165,A -85,B 0,C 180,E1 -18453.146,E2 -18453.146} C_VEL
LIN {X 0,Y 255.847,Z 593.836,A -85,B 0,C 180,E1 -18454.725,E2 -18454.725} C_VEL
LIN {X 0,Y 255.53,Z 590.977,A -85,B 0,C 180,E1 -18457.108,E2 -18457.108} C_VEL
LIN {X 0,Y 255.315,Z 587.032,A -85,B 0,C 180,E1 -18459.505,E2 -18459.505} C_VEL
LIN {X 0,Y 255.397,Z 581.917,A -85,B 0,C 180,E1 -18461.909,E2 -18461.909} C_VEL
LIN {X 0,Y 255.853,Z 575.494,A -85,B 0,C 180,E1 -18464.311,E2 -18464.311} C_VEL
LIN {X 0,Y 256.758,Z 567.669,A -85,B 0,C 180,E1 -18466.661,E2 -18466.661} C_VEL
LIN {X 0,Y 257.881,Z 559.384,A -85,B 0,C 180,E1 -18468.674,E2 -18468.674} C_VEL
LIN {X 0,Y 259.392,Z 549.492,A -85,B 0,C 180,E1 -18470.621,E2 -18470.621} C_VEL
LIN {X 0,Y 260.784,Z 539.816,A -85,B 0,C 180,E1 -18472.164,E2 -18472.164} C_VEL
LIN {X 0,Y 261.359,Z 533.199,A -85,B 0,C 180,E1 -18473.072,E2 -18473.072} C_VEL
LIN {X 0,Y 260.606,Z 520.688,A -85,B 0,C 180,E1 -18474.6,E2 -18474.6} C_VEL
LIN {X 0,Y 259.5,Z 507.387,A -85,B 0,C 180,E1 -18475.89,E2 -18475.89} C_VEL
LIN {X 0,Y 258.715,Z 497.839,A -85,B 0,C 180,E1 -18476.632,E2 -18476.632} C_VEL
LIN {X 0,Y 257.663,Z 482.294,A -85,B 0,C 180,E1 -18477.968,E2 -18477.968} C_VEL
LIN {X 0,Y 256.738,Z 467.125,A -85,B 0,C 180,E1 -18478.993,E2 -18478.993} C_VEL
LIN {X 0,Y 257.941,Z 458.885,A -85,B 0,C 180,E1 -18483.017,E2 -18483.017} C_VEL
LIN {X 0,Y 259.515,Z 449.795,A -85,B 0,C 180,E1 -18487.474,E2 -18487.474} C_VEL
LIN {X 0,Y 260.872,Z 442.598,A -85,B 0,C 180,E1 -18491.033,E2 -18491.033} C_VEL
LIN {X 0,Y 260.709,Z 440.004,A -85,B 0,C 180,E1 -18492.368,E2 -18492.368} C_VEL
LIN {X 0,Y 258.867,Z 431.133,A -85,B 0,C 180,E1 -18497.137,E2 -18497.137} C_VEL
LIN {X 0,Y 257.196,Z 422.764,A -85,B 0,C 180,E1 -18501.883,E2 -18501.883} C_VEL
LIN {X 0,Y 256.132,Z 417.207,A -85,B 0,C 180,E1 -18505.291,E2 -18505.291} C_VEL
LIN {X 0,Y 256.084,Z 417.21,A -85,B 0,C 180,E1 -18508.572,E2 -18508.572} C_VEL
LIN {X 0,Y 256.134,Z 417.203,A -85,B 0,C 180,E1 -18512.196,E2 -18512.196} C_VEL
LIN {X 0,Y 256.158,Z 417.199,A -85,B 0,C 180,E1 -18515.699,E2 -18515.699} C_VEL
LIN {X 0,Y 256.157,Z 417.199,A -85,B 0,C 180,E1 -18519.104,E2 -18519.104} C_VEL
LIN {X 0,Y 256.29,Z 417.181,A -85,B 0,C 180,E1 -18524.085,E2 -18524.085} C_VEL
LIN {X 0,Y 256.301,Z 417.181,A -85,B 0,C 180,E1 -18528.934,E2 -18528.934} C_VEL
LIN {X 0,Y 256.53,Z 417.154,A -85,B 0,C 180,E1 -18532.127,E2 -18532.127} C_VEL
LIN {X 0,Y 256.708,Z 417.133,A -85,B 0,C 180,E1 -18538.432,E2 -18538.432} C_VEL
LIN {X 0,Y 256.708,Z 417.13,A -85,B 0,C 180,E1 -18541.569,E2 -18541.569} C_VEL
LIN {X 0,Y 256.531,Z 417.138,A -85,B 0,C 180,E1 -18547.874,E2 -18547.874} C_VEL
LIN {X 0,Y 256.301,Z 417.172,A -85,B 0,C 180,E1 -18551.067,E2 -18551.067} C_VEL
LIN {X 0,Y 256.291,Z 417.182,A -85,B 0,C 180,E1 -18555.916,E2 -18555.916} C_VEL
LIN {X 0,Y 256.158,Z 417.2,A -85,B 0,C 180,E1 -18560.896,E2 -18560.896} C_VEL
LIN {X 0,Y 256.181,Z 417.198,A -85,B 0,C 180,E1 -18565.14,E2 -18565.14} C_VEL
LIN {X 0,Y 256.097,Z 417.185,A -85,B 0,C 180,E1 -18569.602,E2 -18569.602} C_VEL
LIN {X 0,Y 256.061,Z 417.211,A -85,B 0,C 180,E1 -18573.294,E2 -18573.294} C_VEL
LIN {X 0,Y 256.108,Z 417.193,A -85,B 0,C 180,E1 -18577.272,E2 -18577.272} C_VEL
LIN {X 0,Y 256.05,Z 417.214,A -85,B 0,C 180,E1 -18581.205,E2 -18581.205} C_VEL
LIN {X 0,Y 256.061,Z 417.201,A -85,B 0,C 180,E1 -18585.53,E2 -18585.53} C_VEL
LIN {X 0,Y 256.081,Z 417.211,A -85,B 0,C 180,E1 -18588.805,E2 -18588.805} C_VEL
LIN {X 0,Y 256.153,Z 417.203,A -85,B 0,C 180,E1 -18592.874,E2 -18592.874} C_VEL
LIN {X 0,Y 256.083,Z 417.211,A -85,B 0,C 180,E1 -18596.712,E2 -18596.712} C_VEL
LIN {X 0,Y 256.137,Z 417.204,A -85,B 0,C 180,E1 -18601.407,E2 -18601.407} C_VEL
LIN {X 0,Y 256.194,Z 417.196,A -85,B 0,C 180,E1 -18605.344,E2 -18605.344} C_VEL
LIN {X 0,Y 257.225,Z 420.039,A -85,B 0,C 180,E1 -18605.574,E2 -18605.574} C_VEL
LIN {X 0,Y 262.578,Z 431.878,A -85,B 0,C 180,E1 -18606.766,E2 -18606.766} C_VEL
LIN {X 0,Y 266.983,Z 443.428,A -85,B 0,C 180,E1 -18608.113,E2 -18608.113} C_VEL
LIN {X 0,Y 268.878,Z 449.92,A -85,B 0,C 180,E1 -18608.938,E2 -18608.938} C_VEL
LIN {X 0,Y 267.719,Z 461.813,A -85,B 0,C 180,E1 -18610.248,E2 -18610.248} C_VEL
LIN {X 0,Y 266.293,Z 472.483,A -85,B 0,C 180,E1 -18611.734,E2 -18611.734} C_VEL
LIN {X 0,Y 264.665,Z 482.185,A -85,B 0,C 180,E1 -18613.416,E2 -18613.416} C_VEL
LIN {X 0,Y 262.934,Z 490.947,A -85,B 0,C 180,E1 -18615.292,E2 -18615.292} C_VEL
LIN {X 0,Y 261.265,Z 499.456,A -85,B 0,C 180,E1 -18617.575,E2 -18617.575} C_VEL
LIN {X 0,Y 259.782,Z 506.297,A -85,B 0,C 180,E1 -18619.874,E2 -18619.874} C_VEL
LIN {X 0,Y 258.805,Z 511.701,A -85,B 0,C 180,E1 -18622.198,E2 -18622.198} C_VEL
LIN {X 0,Y 257.827,Z 515.975,A -85,B 0,C 180,E1 -18624.527,E2 -18624.527} C_VEL
LIN {X 0,Y 257.053,Z 519.21,A -85,B 0,C 180,E1 -18626.867,E2 -18626.867} C_VEL
LIN {X 0,Y 256.64,Z 522.006,A -85,B 0,C 180,E1 -18630.002,E2 -18630.002} C_VEL
LIN {X 0,Y 256.628,Z 522.813,A -85,B 0,C 180,E1 -18631.571,E2 -18631.571} C_VEL
LIN {X 0,Y 256.448,Z 523.28,A -85,B 0,C 180,E1 -18634.718,E2 -18634.718} C_VEL
LIN {X 0,Y 256.749,Z 522.924,A -85,B 0,C 180,E1 -18636.288,E2 -18636.288} C_VEL
LIN {X 0,Y 257.249,Z 522.151,A -85,B 0,C 180,E1 -18637.853,E2 -18637.853} C_VEL
LIN {X 0,Y 257.854,Z 520.962,A -85,B 0,C 180,E1 -18639.414,E2 -18639.414} C_VEL
LIN {X 0,Y 258.837,Z 517.928,A -85,B 0,C 180,E1 -18642.179,E2 -18642.179} C_VEL
LIN {X 0,Y 260.194,Z 513.603,A -85,B 0,C 180,E1 -18644.87,E2 -18644.87} C_VEL
LIN {X 0,Y 261.584,Z 508.615,A -85,B 0,C 180,E1 -18647.191,E2 -18647.191} C_VEL
LIN {X 0,Y 263.206,Z 502.311,A -85,B 0,C 180,E1 -18649.499,E2 -18649.499} C_VEL
LIN {X 0,Y 265.236,Z 494.419,A -85,B 0,C 180,E1 -18651.776,E2 -18651.776} C_VEL
LIN {X 0,Y 267.142,Z 486.309,A -85,B 0,C 180,E1 -18653.655,E2 -18653.655} C_VEL
LIN {X 0,Y 269.125,Z 476.281,A -85,B 0,C 180,E1 -18655.525,E2 -18655.525} C_VEL
LIN {X 0,Y 270.958,Z 464.985,A -85,B 0,C 180,E1 -18657.205,E2 -18657.205} C_VEL
LIN {X 0,Y 272.157,Z 455.671,A -85,B 0,C 180,E1 -18658.307,E2 -18658.307} C_VEL
LIN {X 0,Y 270.639,Z 449.745,A -85,B 0,C 180,E1 -18659.17,E2 -18659.17} C_VEL
LIN {X 0,Y 266.469,Z 438.617,A -85,B 0,C 180,E1 -18660.722,E2 -18660.722} C_VEL
LIN {X 0,Y 261.351,Z 427.682,A -85,B 0,C 180,E1 -18662.127,E2 -18662.127} C_VEL
LIN {X 0,Y 257.258,Z 420.213,A -85,B 0,C 180,E1 -18663.033,E2 -18663.033} C_VEL
LIN {X 0,Y 256.14,Z 417.25,A -85,B 0,C 180,E1 -18663.338,E2 -18663.338} C_VEL
LIN {X 0,Y 256.12,Z 417.192,A -85,B 0,C 180,E1 -18667.271,E2 -18667.271} C_VEL
LIN {X 0,Y 256.061,Z 417.215,A -85,B 0,C 180,E1 -18671.204,E2 -18671.204} C_VEL
LIN {X 0,Y 256.05,Z 417.208,A -85,B 0,C 180,E1 -18675.534,E2 -18675.534} C_VEL
LIN {X 0,Y 256.061,Z 417.203,A -85,B 0,C 180,E1 -18678.797,E2 -18678.797} C_VEL
LIN {X 0,Y 256.136,Z 417.176,A -85,B 0,C 180,E1 -18682.868,E2 -18682.868} C_VEL
LIN {X 0,Y 256.074,Z 417.208,A -85,B 0,C 180,E1 -18686.707,E2 -18686.707} C_VEL
LIN {X 0,Y 256.109,Z 417.153,A -85,B 0,C 180,E1 -18690.399,E2 -18690.399} C_VEL
LIN {X 0,Y 256.228,Z 417.351,A -85,B 0,C 180,E1 -18694.467,E2 -18694.467} C_VEL
LIN {X 0,Y 260.128,Z 431.735,A -85,B 0,C 180,E1 -18696.163,E2 -18696.163} C_VEL
LIN {X 0,Y 264.009,Z 445.678,A -85,B 0,C 180,E1 -18698.118,E2 -18698.118} C_VEL
LIN {X 0,Y 263.207,Z 454.962,A -85,B 0,C 180,E1 -18699.442,E2 -18699.442} C_VEL
LIN {X 0,Y 261.466,Z 467.887,A -85,B 0,C 180,E1 -18701.589,E2 -18701.589} C_VEL
LIN {X 0,Y 259.998,Z 479.459,A -85,B 0,C 180,E1 -18703.914,E2 -18703.914} C_VEL
LIN {X 0,Y 258.831,Z 489.149,A -85,B 0,C 180,E1 -18706.255,E2 -18706.255} C_VEL
LIN {X 0,Y 257.752,Z 498.57,A -85,B 0,C 180,E1 -18708.996,E2 -18708.996} C_VEL
LIN {X 0,Y 257.03,Z 506.38,A -85,B 0,C 180,E1 -18711.746,E2 -18711.746} C_VEL
LIN {X 0,Y 256.402,Z 512.779,A -85,B 0,C 180,E1 -18714.494,E2 -18714.494} C_VEL
LIN {X 0,Y 256.379,Z 518.585,A -85,B 0,C 180,E1 -18717.643,E2 -18717.643} C_VEL
LIN {X 0,Y 256.583,Z 521.944,A -85,B 0,C 180,E1 -18720,E2 -18720} C_VEL
LIN {X 0,Y 257.015,Z 525.287,A -85,B 0,C 180,E1 -18723.135,E2 -18723.135} C_VEL
LIN {X 0,Y 257.993,Z 527.332,A -85,B 0,C 180,E1 -18726.255,E2 -18726.255} C_VEL
LIN {X 0,Y 259.582,Z 528.098,A -85,B 0,C 180,E1 -18729.349,E2 -18729.349} C_VEL
LIN {X 0,Y 261.752,Z 527.624,A -85,B 0,C 180,E1 -18732.403,E2 -18732.403} C_VEL
LIN {X 0,Y 264.444,Z 525.946,A -85,B 0,C 180,E1 -18735.412,E2 -18735.412} C_VEL
LIN {X 0,Y 265.454,Z 525.079,A -85,B 0,C 180,E1 -18736.409,E2 -18736.409} C_VEL
LIN {X 0,Y 266.195,Z 524.115,A -85,B 0,C 180,E1 -18737.656,E2 -18737.656} C_VEL
LIN {X 0,Y 265.95,Z 522.008,A -85,B 0,C 180,E1 -18740.61,E2 -18740.61} C_VEL
LIN {X 0,Y 266.538,Z 520.254,A -85,B 0,C 180,E1 -18742.258,E2 -18742.258} C_VEL
LIN {X 0,Y 267.513,Z 519.046,A -85,B 0,C 180,E1 -18743.031,E2 -18743.031} C_VEL
LIN {X 0,Y 272.945,Z 512.816,A -85,B 0,C 180,E1 -18745.959,E2 -18745.959} C_VEL
LIN {X 0,Y 278.675,Z 505.346,A -85,B 0,C 180,E1 -18748.631,E2 -18748.631} C_VEL
LIN {X 0,Y 284.159,Z 497.497,A -85,B 0,C 180,E1 -18750.877,E2 -18750.877} C_VEL
LIN {X 0,Y 290.217,Z 487.938,A -85,B 0,C 180,E1 -18753.101,E2 -18753.101} C_VEL
LIN {X 0,Y 290.484,Z 486.467,A -85,B 0,C 180,E1 -18753.811,E2 -18753.811} C_VEL
LIN {X 0,Y 290.519,Z 485.167,A -85,B 0,C 180,E1 -18754.662,E2 -18754.662} C_VEL
LIN {X 0,Y 290.208,Z 484.311,A -85,B 0,C 180,E1 -18755.535,E2 -18755.535} C_VEL
LIN {X 0,Y 289.254,Z 483.485,A -85,B 0,C 180,E1 -18757.403,E2 -18757.403} C_VEL
LIN {X 0,Y 288.315,Z 483.447,A -85,B 0,C 180,E1 -18759.329,E2 -18759.329} C_VEL
LIN {X 0,Y 287.614,Z 484.2,A -85,B 0,C 180,E1 -18761.281,E2 -18761.281} C_VEL
LIN {X 0,Y 287.005,Z 486.016,A -85,B 0,C 180,E1 -18763.286,E2 -18763.286} C_VEL
LIN {X 0,Y 286.492,Z 488.075,A -85,B 0,C 180,E1 -18764.649,E2 -18764.649} C_VEL
LIN {X 0,Y 284.588,Z 493.789,A -85,B 0,C 180,E1 -18766.744,E2 -18766.744} C_VEL
LIN {X 0,Y 282.807,Z 500.316,A -85,B 0,C 180,E1 -18768.778,E2 -18768.778} C_VEL
LIN {X 0,Y 280.823,Z 507.987,A -85,B 0,C 180,E1 -18770.879,E2 -18770.879} C_VEL
LIN {X 0,Y 277.755,Z 518.765,A -85,B 0,C 180,E1 -18773.513,E2 -18773.513} C_VEL
LIN {X 0,Y 274.488,Z 528.493,A -85,B 0,C 180,E1 -18775.715,E2 -18775.715} C_VEL
LIN {X 0,Y 270.436,Z 537.926,A -85,B 0,C 180,E1 -18777.807,E2 -18777.807} C_VEL
LIN {X 0,Y 265.823,Z 548.079,A -85,B 0,C 180,E1 -18780.281,E2 -18780.281} C_VEL
LIN {X 0,Y 262.429,Z 554.735,A -85,B 0,C 180,E1 -18782.052,E2 -18782.052} C_VEL
LIN {X 0,Y 257.52,Z 564.141,A -85,B 0,C 180,E1 -18784.974,E2 -18784.974} C_VEL
LIN {X 0,Y 253.565,Z 572.135,A -85,B 0,C 180,E1 -18788.025,E2 -18788.025} C_VEL
LIN {X 0,Y 250.765,Z 578.81,A -85,B 0,C 180,E1 -18791.196,E2 -18791.196} C_VEL
LIN {X 0,Y 248.87,Z 584.222,A -85,B 0,C 180,E1 -18794.437,E2 -18794.437} C_VEL
LIN {X 0,Y 248.092,Z 587.461,A -85,B 0,C 180,E1 -18796.9,E2 -18796.9} C_VEL
LIN {X 0,Y 247.82,Z 590.751,A -85,B 0,C 180,E1 -18800.201,E2 -18800.201} C_VEL
LIN {X 0,Y 248.318,Z 592.815,A -85,B 0,C 180,E1 -18803.498,E2 -18803.498} C_VEL
LIN {X 0,Y 248.553,Z 594.111,A -85,B 0,C 180,E1 -18805.132,E2 -18805.132} C_VEL
LIN {X 0,Y 249.214,Z 595.468,A -85,B 0,C 180,E1 -18808.382,E2 -18808.382} C_VEL
LIN {X 0,Y 249.545,Z 595.52,A -85,B 0,C 180,E1 -18809.998,E2 -18809.998} C_VEL
LIN {X 0,Y 249.276,Z 595.066,A -85,B 0,C 180,E1 -18811.614,E2 -18811.614} C_VEL
LIN {X 0,Y 248.771,Z 592.787,A -85,B 0,C 180,E1 -18814.86,E2 -18814.86} C_VEL
LIN {X 0,Y 248.53,Z 590.999,A -85,B 0,C 180,E1 -18816.493,E2 -18816.493} C_VEL
LIN {X 0,Y 248.285,Z 587.406,A -85,B 0,C 180,E1 -18818.955,E2 -18818.955} C_VEL
LIN {X 0,Y 248.267,Z 582.675,A -85,B 0,C 180,E1 -18821.427,E2 -18821.427} C_VEL
LIN {X 0,Y 248.765,Z 575.521,A -85,B 0,C 180,E1 -18824.31,E2 -18824.31} C_VEL
LIN {X 0,Y 249.762,Z 567.286,A -85,B 0,C 180,E1 -18826.919,E2 -18826.919} C_VEL
LIN {X 0,Y 251.062,Z 558.188,A -85,B 0,C 180,E1 -18829.201,E2 -18829.201} C_VEL
LIN {X 0,Y 252.613,Z 548.256,A -85,B 0,C 180,E1 -18831.201,E2 -18831.201} C_VEL
LIN {X 0,Y 254.264,Z 537.538,A -85,B 0,C 180,E1 -18832.927,E2 -18832.927} C_VEL
LIN {X 0,Y 254.479,Z 532.783,A -85,B 0,C 180,E1 -18833.605,E2 -18833.605} C_VEL
LIN {X 0,Y 253.791,Z 520.256,A -85,B 0,C 180,E1 -18835.197,E2 -18835.197} C_VEL
LIN {X 0,Y 252.809,Z 507.16,A -85,B 0,C 180,E1 -18836.519,E2 -18836.519} C_VEL
LIN {X 0,Y 251.615,Z 493.768,A -85,B 0,C 180,E1 -18837.523,E2 -18837.523} C_VEL
LIN {X 0,Y 250.89,Z 485.975,A -85,B 0,C 180,E1 -18837.98,E2 -18837.98} C_VEL
LIN {X 0,Y 249.95,Z 470.523,A -85,B 0,C 180,E1 -18839.115,E2 -18839.115} C_VEL
LIN {X 0,Y 249.768,Z 466.16,A -85,B 0,C 180,E1 -18839.429,E2 -18839.429} C_VEL
LIN {X 0,Y 251.148,Z 457.053,A -85,B 0,C 180,E1 -18844.03,E2 -18844.03} C_VEL
LIN {X 0,Y 252.722,Z 448.574,A -85,B 0,C 180,E1 -18848.339,E2 -18848.339} C_VEL
LIN {X 0,Y 253.655,Z 444.105,A -85,B 0,C 180,E1 -18850.613,E2 -18850.613} C_VEL
LIN {X 0,Y 253.692,Z 441.077,A -85,B 0,C 180,E1 -18852.194,E2 -18852.194} C_VEL
LIN {X 0,Y 252.056,Z 433.329,A -85,B 0,C 180,E1 -18856.461,E2 -18856.461} C_VEL
LIN {X 0,Y 250.532,Z 425.684,A -85,B 0,C 180,E1 -18860.863,E2 -18860.863} C_VEL
LIN {X 0,Y 249.096,Z 418.129,A -85,B 0,C 180,E1 -18865.441,E2 -18865.441} C_VEL
LIN {X 0,Y 249.043,Z 418.086,A -85,B 0,C 180,E1 -18869.472,E2 -18869.472} C_VEL
LIN {X 0,Y 249.066,Z 418.087,A -85,B 0,C 180,E1 -18873.162,E2 -18873.162} C_VEL
LIN {X 0,Y 249.07,Z 418.083,A -85,B 0,C 180,E1 -18876.732,E2 -18876.732} C_VEL
LIN {X 0,Y 249.101,Z 418.074,A -85,B 0,C 180,E1 -18880.211,E2 -18880.211} C_VEL
LIN {X 0,Y 249.233,Z 418.061,A -85,B 0,C 180,E1 -18883.622,E2 -18883.622} C_VEL
LIN {X 0,Y 249.244,Z 418.063,A -85,B 0,C 180,E1 -18888.617,E2 -18888.617} C_VEL
LIN {X 0,Y 249.472,Z 418.033,A -85,B 0,C 180,E1 -18891.903,E2 -18891.903} C_VEL
LIN {X 0,Y 249.432,Z 418.038,A -85,B 0,C 180,E1 -18896.77,E2 -18896.77} C_VEL
LIN {X 0,Y 249.727,Z 417.998,A -85,B 0,C 180,E1 -18900,E2 -18900} C_VEL
LIN {X 0,Y 249.433,Z 418.04,A -85,B 0,C 180,E1 -18903.231,E2 -18903.231} C_VEL
LIN {X 0,Y 249.472,Z 418.013,A -85,B 0,C 180,E1 -18908.098,E2 -18908.098} C_VEL
LIN {X 0,Y 249.245,Z 418.053,A -85,B 0,C 180,E1 -18911.384,E2 -18911.384} C_VEL
LIN {X 0,Y 249.234,Z 418.062,A -85,B 0,C 180,E1 -18916.379,E2 -18916.379} C_VEL
LIN {X 0,Y 249.079,Z 418.078,A -85,B 0,C 180,E1 -18921.519,E2 -18921.519} C_VEL
LIN {X 0,Y 249.123,Z 418.076,A -85,B 0,C 180,E1 -18925.484,E2 -18925.484} C_VEL
LIN {X 0,Y 249.066,Z 418.061,A -85,B 0,C 180,E1 -18928.991,E2 -18928.991} C_VEL
LIN {X 0,Y 249.024,Z 418.083,A -85,B 0,C 180,E1 -18932.427,E2 -18932.427} C_VEL
LIN {X 0,Y 249.042,Z 418.08,A -85,B 0,C 180,E1 -18936.344,E2 -18936.344} C_VEL
LIN {X 0,Y 249.001,Z 418.088,A -85,B 0,C 180,E1 -18940.48,E2 -18940.48} C_VEL
LIN {X 0,Y 249.005,Z 418.08,A -85,B 0,C 180,E1 -18944.88,E2 -18944.88} C_VEL
LIN {X 0,Y 249.036,Z 418.087,A -85,B 0,C 180,E1 -18947.37,E2 -18947.37} C_VEL
LIN {X 0,Y 249.045,Z 418.081,A -85,B 0,C 180,E1 -18951.626,E2 -18951.626} C_VEL
LIN {X 0,Y 249.059,Z 418.085,A -85,B 0,C 180,E1 -18955.644,E2 -18955.644} C_VEL
LIN {X 0,Y 249.05,Z 418.08,A -85,B 0,C 180,E1 -18959.475,E2 -18959.475} C_VEL
LIN {X 0,Y 249.073,Z 418.083,A -85,B 0,C 180,E1 -18963.165,E2 -18963.165} C_VEL
LIN {X 0,Y 249.116,Z 418.079,A -85,B 0,C 180,E1 -18964.527,E2 -18964.527} C_VEL
LIN {X 0,Y 250.279,Z 421.127,A -85,B 0,C 180,E1 -18964.795,E2 -18964.795} C_VEL
LIN {X 0,Y 255.557,Z 432.471,A -85,B 0,C 180,E1 -18966.003,E2 -18966.003} C_VEL
LIN {X 0,Y 259.878,Z 443.606,A -85,B 0,C 180,E1 -18967.349,E2 -18967.349} C_VEL
LIN {X 0,Y 262.27,Z 451.432,A -85,B 0,C 180,E1 -18968.388,E2 -18968.388} C_VEL
LIN {X 0,Y 261.137,Z 463.159,A -85,B 0,C 180,E1 -18969.728,E2 -18969.728} C_VEL
LIN {X 0,Y 259.65,Z 473.704,A -85,B 0,C 180,E1 -18971.239,E2 -18971.239} C_VEL
LIN {X 0,Y 257.971,Z 483.4,A -85,B 0,C 180,E1 -18972.972,E2 -18972.972} C_VEL
LIN {X 0,Y 256.163,Z 492.129,A -85,B 0,C 180,E1 -18974.894,E2 -18974.894} C_VEL
LIN {X 0,Y 254.427,Z 500.609,A -85,B 0,C 180,E1 -18977.235,E2 -18977.235} C_VEL
LIN {X 0,Y 252.909,Z 507.409,A -85,B 0,C 180,E1 -18979.596,E2 -18979.596} C_VEL
LIN {X 0,Y 251.857,Z 512.794,A -85,B 0,C 180,E1 -18981.982,E2 -18981.982} C_VEL
LIN {X 0,Y 250.838,Z 517.049,A -85,B 0,C 180,E1 -18984.374,E2 -18984.374} C_VEL
LIN {X 0,Y 250.039,Z 520.264,A -85,B 0,C 180,E1 -18986.779,E2 -18986.779} C_VEL
LIN {X 0,Y 249.614,Z 523.042,A -85,B 0,C 180,E1 -18990.002,E2 -18990.002} C_VEL
LIN {X 0,Y 249.604,Z 523.831,A -85,B 0,C 180,E1 -18991.615,E2 -18991.615} C_VEL
LIN {X 0,Y 249.436,Z 524.281,A -85,B 0,C 180,E1 -18994.851,E2 -18994.851} C_VEL
LIN {X 0,Y 249.758,Z 523.915,A -85,B 0,C 180,E1 -18996.464,E2 -18996.464} C_VEL
LIN {X 0,Y 250.285,Z 523.122,A -85,B 0,C 180,E1 -18998.073,E2 -18998.073} C_VEL
LIN {X 0,Y 250.919,Z 521.925,A -85,B 0,C 180,E1 -18999.676,E2 -18999.676} C_VEL
LIN {X 0,Y 251.968,Z 518.874,A -85,B 0,C 180,E1 -19002.514,E2 -19002.514} C_VEL
LIN {X 0,Y 253.39,Z 514.517,A -85,B 0,C 180,E1 -19005.279,E2 -19005.279} C_VEL
LIN {X 0,Y 254.865,Z 509.502,A -85,B 0,C 180,E1 -19007.659,E2 -19007.659} C_VEL
LIN {X 0,Y 256.575,Z 503.172,A -85,B 0,C 180,E1 -19010.024,E2 -19010.024} C_VEL
LIN {X 0,Y 258.704,Z 495.249,A -85,B 0,C 180,E1 -19012.355,E2 -19012.355} C_VEL
LIN {X 0,Y 260.706,Z 487.095,A -85,B 0,C 180,E1 -19014.276,E2 -19014.276} C_VEL
LIN {X 0,Y 262.781,Z 477.007,A -85,B 0,C 180,E1 -19016.188,E2 -19016.188} C_VEL
LIN {X 0,Y 264.691,Z 465.648,A -85,B 0,C 180,E1 -19017.904,E2 -19017.904} C_VEL
LIN {X 0,Y 265.766,Z 456.891,A -85,B 0,C 180,E1 -19018.972,E2 -19018.972} C_VEL
LIN {X 0,Y 262.389,Z 446.396,A -85,B 0,C 180,E1 -19020.593,E2 -19020.593} C_VEL
LIN {X 0,Y 257.819,Z 435.485,A -85,B 0,C 180,E1 -19022.14,E2 -19022.14} C_VEL
LIN {X 0,Y 252.231,Z 424.612,A -85,B 0,C 180,E1 -19023.577,E2 -19023.577} C_VEL
LIN {X 0,Y 250.332,Z 421.293,A -85,B 0,C 180,E1 -19024.002,E2 -19024.002} C_VEL
LIN {X 0,Y 249.206,Z 418.766,A -85,B 0,C 180,E1 -19024.262,E2 -19024.262} C_VEL
LIN {X 0,Y 249.093,Z 418.118,A -85,B 0,C 180,E1 -19024.399,E2 -19024.399} C_VEL
LIN {X 0,Y 249.031,Z 418.069,A -85,B 0,C 180,E1 -19028.381,E2 -19028.381} C_VEL
LIN {X 0,Y 249.015,Z 418.087,A -85,B 0,C 180,E1 -19032.793,E2 -19032.793} C_VEL
LIN {X 0,Y 249.016,Z 418.092,A -85,B 0,C 180,E1 -19037.362,E2 -19037.362} C_VEL
LIN {X 0,Y 249.031,Z 418.049,A -85,B 0,C 180,E1 -19041.62,E2 -19041.62} C_VEL
LIN {X 0,Y 249.05,Z 418.089,A -85,B 0,C 180,E1 -19045.64,E2 -19045.64} C_VEL
LIN {X 0,Y 249.053,Z 418.034,A -85,B 0,C 180,E1 -19049.473,E2 -19049.473} C_VEL
LIN {X 0,Y 249.114,Z 418.068,A -85,B 0,C 180,E1 -19053.912,E2 -19053.912} C_VEL
LIN {X 0,Y 249.162,Z 418.153,A -85,B 0,C 180,E1 -19054.107,E2 -19054.107} C_VEL
LIN {X 0,Y 252.704,Z 431.31,A -85,B 0,C 180,E1 -19055.678,E2 -19055.678} C_VEL
LIN {X 0,Y 256.52,Z 444.993,A -85,B 0,C 180,E1 -19057.622,E2 -19057.622} C_VEL
LIN {X 0,Y 257.114,Z 447.686,A -85,B 0,C 180,E1 -19058.029,E2 -19058.029} C_VEL
LIN {X 0,Y 255.634,Z 460.124,A -85,B 0,C 180,E1 -19059.9,E2 -19059.9} C_VEL
LIN {X 0,Y 253.822,Z 473.075,A -85,B 0,C 180,E1 -19062.267,E2 -19062.267} C_VEL
LIN {X 0,Y 252.491,Z 483.945,A -85,B 0,C 180,E1 -19064.666,E2 -19064.666} C_VEL
LIN {X 0,Y 251.189,Z 494.529,A -85,B 0,C 180,E1 -19067.476,E2 -19067.476} C_VEL
LIN {X 0,Y 250.298,Z 503.218,A -85,B 0,C 180,E1 -19070.301,E2 -19070.301} C_VEL
LIN {X 0,Y 249.76,Z 509.495,A -85,B 0,C 180,E1 -19072.725,E2 -19072.725} C_VEL
LIN {X 0,Y 249.16,Z 516.292,A -85,B 0,C 180,E1 -19075.956,E2 -19075.956} C_VEL
LIN {X 0,Y 249.456,Z 521.546,A -85,B 0,C 180,E1 -19079.192,E2 -19079.192} C_VEL
LIN {X 0,Y 249.665,Z 524.596,A -85,B 0,C 180,E1 -19081.613,E2 -19081.613} C_VEL
LIN {X 0,Y 250.452,Z 527.486,A -85,B 0,C 180,E1 -19084.829,E2 -19084.829} C_VEL
LIN {X 0,Y 251.801,Z 529.106,A -85,B 0,C 180,E1 -19088.022,E2 -19088.022} C_VEL
LIN {X 0,Y 253.799,Z 529.468,A -85,B 0,C 180,E1 -19091.177,E2 -19091.177} C_VEL
LIN {X 0,Y 256.38,Z 528.621,A -85,B 0,C 180,E1 -19094.283,E2 -19094.283} C_VEL
LIN {X 0,Y 259.471,Z 526.6,A -85,B 0,C 180,E1 -19097.334,E2 -19097.334} C_VEL
LIN {X 0,Y 263.295,Z 523.324,A -85,B 0,C 180,E1 -19100.304,E2 -19100.304} C_VEL
LIN {X 0,Y 267.513,Z 519.046,A -85,B 0,C 180,E1 -19103.031,E2 -19103.031} C_VEL
LIN {X 0,Y 268.917,Z 517.215,A -85,B 0,C 180,E1 -19104.194,E2 -19104.194} C_VEL
LIN {X 0,Y 270.856,Z 512.086,A -85,B 0,C 180,E1 -19107.796,E2 -19107.796} C_VEL
LIN {X 0,Y 272.312,Z 509.799,A -85,B 0,C 180,E1 -19108.897,E2 -19108.897} C_VEL
LIN {X 0,Y 273.028,Z 508.91,A -85,B 0,C 180,E1 -19109.233,E2 -19109.233} C_VEL
LIN {X 0,Y 279.685,Z 500.235,A -85,B 0,C 180,E1 -19111.849,E2 -19111.849} C_VEL
LIN {X 0,Y 284.777,Z 493.021,A -85,B 0,C 180,E1 -19113.599,E2 -19113.599} C_VEL
LIN {X 0,Y 285.652,Z 491.296,A -85,B 0,C 180,E1 -19114.201,E2 -19114.201} C_VEL
LIN {X 0,Y 285.557,Z 489.666,A -85,B 0,C 180,E1 -19115.689,E2 -19115.689} C_VEL
LIN {X 0,Y 284.465,Z 489.011,A -85,B 0,C 180,E1 -19118.144,E2 -19118.144} C_VEL
LIN {X 0,Y 283.699,Z 489.365,A -85,B 0,C 180,E1 -19120.097,E2 -19120.097} C_VEL
LIN {X 0,Y 283.032,Z 490.672,A -85,B 0,C 180,E1 -19122.101,E2 -19122.101} C_VEL
LIN {X 0,Y 282.481,Z 492.62,A -85,B 0,C 180,E1 -19123.819,E2 -19123.819} C_VEL
LIN {X 0,Y 281.286,Z 495.607,A -85,B 0,C 180,E1 -19125.105,E2 -19125.105} C_VEL
LIN {X 0,Y 278.295,Z 504.045,A -85,B 0,C 180,E1 -19127.959,E2 -19127.959} C_VEL
LIN {X 0,Y 275.96,Z 511.261,A -85,B 0,C 180,E1 -19130.053,E2 -19130.053} C_VEL
LIN {X 0,Y 272.484,Z 521.41,A -85,B 0,C 180,E1 -19132.69,E2 -19132.69} C_VEL
LIN {X 0,Y 268.916,Z 530.545,A -85,B 0,C 180,E1 -19134.902,E2 -19134.902} C_VEL
LIN {X 0,Y 264.605,Z 539.505,A -85,B 0,C 180,E1 -19137.009,E2 -19137.009} C_VEL
LIN {X 0,Y 259.151,Z 550.417,A -85,B 0,C 180,E1 -19139.885,E2 -19139.885} C_VEL
LIN {X 0,Y 254.021,Z 559.082,A -85,B 0,C 180,E1 -19142.434,E2 -19142.434} C_VEL
LIN {X 0,Y 248.956,Z 568.361,A -85,B 0,C 180,E1 -19145.835,E2 -19145.835} C_VEL
LIN {X 0,Y 245.321,Z 575.345,A -85,B 0,C 180,E1 -19149.015,E2 -19149.015} C_VEL
LIN {X 0,Y 242.794,Z 581.232,A -85,B 0,C 180,E1 -19152.391,E2 -19152.391} C_VEL
LIN {X 0,Y 241.59,Z 584.648,A -85,B 0,C 180,E1 -19154.82,E2 -19154.82} C_VEL
LIN {X 0,Y 240.84,Z 588.318,A -85,B 0,C 180,E1 -19158.212,E2 -19158.212} C_VEL
LIN {X 0,Y 240.901,Z 590.79,A -85,B 0,C 180,E1 -19161.611,E2 -19161.611} C_VEL
LIN {X 0,Y 241.215,Z 591.789,A -85,B 0,C 180,E1 -19163.306,E2 -19163.306} C_VEL
LIN {X 0,Y 241.474,Z 593.12,A -85,B 0,C 180,E1 -19164.989,E2 -19164.989} C_VEL
LIN {X 0,Y 242.168,Z 594.464,A -85,B 0,C 180,E1 -19168.335,E2 -19168.335} C_VEL
LIN {X 0,Y 242.512,Z 594.511,A -85,B 0,C 180,E1 -19169.998,E2 -19169.998} C_VEL
LIN {X 0,Y 242.235,Z 594.044,A -85,B 0,C 180,E1 -19171.661,E2 -19171.661} C_VEL
LIN {X 0,Y 241.681,Z 591.736,A -85,B 0,C 180,E1 -19175.003,E2 -19175.003} C_VEL
LIN {X 0,Y 241.289,Z 588.222,A -85,B 0,C 180,E1 -19177.982,E2 -19177.982} C_VEL
LIN {X 0,Y 241.178,Z 583.27,A -85,B 0,C 180,E1 -19180.916,E2 -19180.916} C_VEL
LIN {X 0,Y 241.581,Z 576.634,A -85,B 0,C 180,E1 -19183.885,E2 -19183.885} C_VEL
LIN {X 0,Y 242.409,Z 569.435,A -85,B 0,C 180,E1 -19186.418,E2 -19186.418} C_VEL
LIN {X 0,Y 243.721,Z 560.449,A -85,B 0,C 180,E1 -19188.928,E2 -19188.928} C_VEL
LIN {X 0,Y 245.462,Z 550.286,A -85,B 0,C 180,E1 -19191.189,E2 -19191.189} C_VEL
LIN {X 0,Y 247.123,Z 539.896,A -85,B 0,C 180,E1 -19193.017,E2 -19193.017} C_VEL
LIN {X 0,Y 247.622,Z 533.698,A -85,B 0,C 180,E1 -19193.962,E2 -19193.962} C_VEL
LIN {X 0,Y 247.136,Z 522.803,A -85,B 0,C 180,E1 -19195.467,E2 -19195.467} C_VEL
LIN {X 0,Y 246.302,Z 510.085,A -85,B 0,C 180,E1 -19196.891,E2 -19196.891} C_VEL
LIN {X 0,Y 245.327,Z 496.836,A -85,B 0,C 180,E1 -19198.008,E2 -19198.008} C_VEL
LIN {X 0,Y 244.025,Z 483.057,A -85,B 0,C 180,E1 -19198.833,E2 -19198.833} C_VEL
LIN {X 0,Y 243.051,Z 471.826,A -85,B 0,C 180,E1 -19199.379,E2 -19199.379} C_VEL
LIN {X 0,Y 242.835,Z 464.826,A -85,B 0,C 180,E1 -19200.176,E2 -19200.176} C_VEL
LIN {X 0,Y 244.071,Z 457.011,A -85,B 0,C 180,E1 -19204.156,E2 -19204.156} C_VEL
LIN {X 0,Y 245.463,Z 449.695,A -85,B 0,C 180,E1 -19207.991,E2 -19207.991} C_VEL
LIN {X 0,Y 246.618,Z 444.082,A -85,B 0,C 180,E1 -19210.95,E2 -19210.95} C_VEL
LIN {X 0,Y 246.636,Z 441.783,A -85,B 0,C 180,E1 -19212.194,E2 -19212.194} C_VEL
LIN {X 0,Y 245.012,Z 434.161,A -85,B 0,C 180,E1 -19216.495,E2 -19216.495} C_VEL
LIN {X 0,Y 243.412,Z 426.188,A -85,B 0,C 180,E1 -19221.217,E2 -19221.217} C_VEL
LIN {X 0,Y 242.101,Z 419.295,A -85,B 0,C 180,E1 -19225.524,E2 -19225.524} C_VEL
LIN {X 0,Y 241.989,Z 418.966,A -85,B 0,C 180,E1 -19226.009,E2 -19226.009} C_VEL
LIN {X 0,Y 242.028,Z 418.958,A -85,B 0,C 180,E1 -19230.586,E2 -19230.586} C_VEL
LIN {X 0,Y 242.059,Z 418.955,A -85,B 0,C 180,E1 -19234.182,E2 -19234.182} C_VEL
LIN {X 0,Y 242.044,Z 418.959,A -85,B 0,C 180,E1 -19238.297,E2 -19238.297} C_VEL
LIN {X 0,Y 242.154,Z 418.944,A -85,B 0,C 180,E1 -19243.278,E2 -19243.278} C_VEL
LIN {X 0,Y 242.178,Z 418.942,A -85,B 0,C 180,E1 -19248.28,E2 -19248.28} C_VEL
LIN {X 0,Y 242.418,Z 418.912,A -85,B 0,C 180,E1 -19251.666,E2 -19251.666} C_VEL
LIN {X 0,Y 242.253,Z 418.929,A -85,B 0,C 180,E1 -19255.007,E2 -19255.007} C_VEL
LIN {X 0,Y 242.63,Z 418.887,A -85,B 0,C 180,E1 -19258.341,E2 -19258.341} C_VEL
LIN {X 0,Y 242.631,Z 418.884,A -85,B 0,C 180,E1 -19261.66,E2 -19261.66} C_VEL
LIN {X 0,Y 242.42,Z 418.899,A -85,B 0,C 180,E1 -19266.74,E2 -19266.74} C_VEL
LIN {X 0,Y 242.305,Z 418.905,A -85,B 0,C 180,E1 -19270.023,E2 -19270.023} C_VEL
LIN {X 0,Y 242.159,Z 418.945,A -85,B 0,C 180,E1 -19275.142,E2 -19275.142} C_VEL
LIN {X 0,Y 242.065,Z 418.956,A -85,B 0,C 180,E1 -19278.625,E2 -19278.625} C_VEL
LIN {X 0,Y 242.005,Z 418.959,A -85,B 0,C 180,E1 -19282.181,E2 -19282.181} C_VEL
LIN {X 0,Y 242.059,Z 418.956,A -85,B 0,C 180,E1 -19285.84,E2 -19285.84} C_VEL
LIN {X 0,Y 242,Z 418.938,A -85,B 0,C 180,E1 -19289.585,E2 -19289.585} C_VEL
LIN {X 0,Y 241.974,Z 418.966,A -85,B 0,C 180,E1 -19293.494,E2 -19293.494} C_VEL
LIN {X 0,Y 241.983,Z 418.95,A -85,B 0,C 180,E1 -19297.584,E2 -19297.584} C_VEL
LIN {X 0,Y 241.934,Z 418.973,A -85,B 0,C 180,E1 -19301.924,E2 -19301.924} C_VEL
LIN {X 0,Y 241.948,Z 418.964,A -85,B 0,C 180,E1 -19306.569,E2 -19306.569} C_VEL
LIN {X 0,Y 241.978,Z 418.96,A -85,B 0,C 180,E1 -19310.288,E2 -19310.288} C_VEL
LIN {X 0,Y 242.034,Z 418.96,A -85,B 0,C 180,E1 -19314.5,E2 -19314.5} C_VEL
LIN {X 0,Y 241.974,Z 418.963,A -85,B 0,C 180,E1 -19318.482,E2 -19318.482} C_VEL
LIN {X 0,Y 242.008,Z 418.96,A -85,B 0,C 180,E1 -19322.315,E2 -19322.315} C_VEL
LIN {X 0,Y 242.049,Z 418.962,A -85,B 0,C 180,E1 -19323.676,E2 -19323.676} C_VEL
LIN {X 0,Y 243.069,Z 421.82,A -85,B 0,C 180,E1 -19323.915,E2 -19323.915} C_VEL
LIN {X 0,Y 247.95,Z 431.764,A -85,B 0,C 180,E1 -19325.031,E2 -19325.031} C_VEL
LIN {X 0,Y 252.212,Z 442.308,A -85,B 0,C 180,E1 -19326.335,E2 -19326.335} C_VEL
LIN {X 0,Y 255.434,Z 452.201,A -85,B 0,C 180,E1 -19327.695,E2 -19327.695} C_VEL
LIN {X 0,Y 255.783,Z 454.31,A -85,B 0,C 180,E1 -19327.979,E2 -19327.979} C_VEL
LIN {X 0,Y 254.369,Z 465.997,A -85,B 0,C 180,E1 -19329.376,E2 -19329.376} C_VEL
LIN {X 0,Y 252.682,Z 476.749,A -85,B 0,C 180,E1 -19331.028,E2 -19331.028} C_VEL
LIN {X 0,Y 250.91,Z 486.492,A -85,B 0,C 180,E1 -19332.898,E2 -19332.898} C_VEL
LIN {X 0,Y 249.071,Z 494.876,A -85,B 0,C 180,E1 -19334.872,E2 -19334.872} C_VEL
LIN {X 0,Y 247.359,Z 502.972,A -85,B 0,C 180,E1 -19337.282,E2 -19337.282} C_VEL
LIN {X 0,Y 246.031,Z 508.522,A -85,B 0,C 180,E1 -19339.301,E2 -19339.301} C_VEL
LIN {X 0,Y 244.913,Z 513.888,A -85,B 0,C 180,E1 -19341.753,E2 -19341.753} C_VEL
LIN {X 0,Y 243.85,Z 518.123,A -85,B 0,C 180,E1 -19344.212,E2 -19344.212} C_VEL
LIN {X 0,Y 243.026,Z 521.319,A -85,B 0,C 180,E1 -19346.686,E2 -19346.686} C_VEL
LIN {X 0,Y 242.588,Z 524.079,A -85,B 0,C 180,E1 -19350.002,E2 -19350.002} C_VEL
LIN {X 0,Y 242.579,Z 524.849,A -85,B 0,C 180,E1 -19351.662,E2 -19351.662} C_VEL
LIN {X 0,Y 242.427,Z 525.281,A -85,B 0,C 180,E1 -19354.991,E2 -19354.991} C_VEL
LIN {X 0,Y 242.77,Z 524.905,A -85,B 0,C 180,E1 -19356.651,E2 -19356.651} C_VEL
LIN {X 0,Y 243.326,Z 524.094,A -85,B 0,C 180,E1 -19358.305,E2 -19358.305} C_VEL
LIN {X 0,Y 243.99,Z 522.887,A -85,B 0,C 180,E1 -19359.954,E2 -19359.954} C_VEL
LIN {X 0,Y 245.11,Z 519.819,A -85,B 0,C 180,E1 -19362.867,E2 -19362.867} C_VEL
LIN {X 0,Y 246.604,Z 515.428,A -85,B 0,C 180,E1 -19365.71,E2 -19365.71} C_VEL
LIN {X 0,Y 248.165,Z 510.389,A -85,B 0,C 180,E1 -19368.152,E2 -19368.152} C_VEL
LIN {X 0,Y 249.966,Z 504.033,A -85,B 0,C 180,E1 -19370.578,E2 -19370.578} C_VEL
LIN {X 0,Y 252.2,Z 496.08,A -85,B 0,C 180,E1 -19372.965,E2 -19372.965} C_VEL
LIN {X 0,Y 254.29,Z 487.879,A -85,B 0,C 180,E1 -19374.929,E2 -19374.929} C_VEL
LIN {X 0,Y 256.476,Z 477.735,A -85,B 0,C 180,E1 -19376.882,E2 -19376.882} C_VEL
LIN {X 0,Y 258.381,Z 466.784,A -85,B 0,C 180,E1 -19378.573,E2 -19378.573} C_VEL
LIN {X 0,Y 259.437,Z 459.1,A -85,B 0,C 180,E1 -19379.534,E2 -19379.534} C_VEL
LIN {X 0,Y 256.456,Z 449.61,A -85,B 0,C 180,E1 -19381.086,E2 -19381.086} C_VEL
LIN {X 0,Y 252.295,Z 439.279,A -85,B 0,C 180,E1 -19382.656,E2 -19382.656} C_VEL
LIN {X 0,Y 246.796,Z 428.278,A -85,B 0,C 180,E1 -19384.233,E2 -19384.233} C_VEL
LIN {X 0,Y 243.5,Z 422.512,A -85,B 0,C 180,E1 -19385.018,E2 -19385.018} C_VEL
LIN {X 0,Y 242.177,Z 419.863,A -85,B 0,C 180,E1 -19385.33,E2 -19385.33} C_VEL
LIN {X 0,Y 242.043,Z 419.12,A -85,B 0,C 180,E1 -19385.503,E2 -19385.503} C_VEL
LIN {X 0,Y 241.962,Z 418.958,A -85,B 0,C 180,E1 -19389.72,E2 -19389.72} C_VEL
LIN {X 0,Y 241.932,Z 418.975,A -85,B 0,C 180,E1 -19394.204,E2 -19394.204} C_VEL
LIN {X 0,Y 241.94,Z 418.97,A -85,B 0,C 180,E1 -19398.077,E2 -19398.077} C_VEL
LIN {X 0,Y 241.994,Z 418.93,A -85,B 0,C 180,E1 -19402.418,E2 -19402.418} C_VEL
LIN {X 0,Y 241.987,Z 418.963,A -85,B 0,C 180,E1 -19406.508,E2 -19406.508} C_VEL
LIN {X 0,Y 242.02,Z 418.906,A -85,B 0,C 180,E1 -19410.597,E2 -19410.597} C_VEL
LIN {X 0,Y 242.069,Z 418.944,A -85,B 0,C 180,E1 -19413.738,E2 -19413.738} C_VEL
LIN {X 0,Y 245.562,Z 431.894,A -85,B 0,C 180,E1 -19415.326,E2 -19415.326} C_VEL
LIN {X 0,Y 249.006,Z 444.386,A -85,B 0,C 180,E1 -19417.124,E2 -19417.124} C_VEL
LIN {X 0,Y 249.91,Z 447.743,A -85,B 0,C 180,E1 -19417.656,E2 -19417.656} C_VEL
LIN {X 0,Y 249.746,Z 452.004,A -85,B 0,C 180,E1 -19418.288,E2 -19418.288} C_VEL
LIN {X 0,Y 248.085,Z 464.632,A -85,B 0,C 180,E1 -19420.341,E2 -19420.341} C_VEL
LIN {X 0,Y 246.457,Z 476.09,A -85,B 0,C 180,E1 -19422.577,E2 -19422.577} C_VEL
LIN {X 0,Y 245.186,Z 486.647,A -85,B 0,C 180,E1 -19425.05,E2 -19425.05} C_VEL
LIN {X 0,Y 243.916,Z 496.896,A -85,B 0,C 180,E1 -19427.942,E2 -19427.942} C_VEL
LIN {X 0,Y 243.057,Z 505.395,A -85,B 0,C 180,E1 -19430.849,E2 -19430.849} C_VEL
LIN {X 0,Y 242.465,Z 511.503,A -85,B 0,C 180,E1 -19433.342,E2 -19433.342} C_VEL
LIN {X 0,Y 242.092,Z 516.676,A -85,B 0,C 180,E1 -19435.838,E2 -19435.838} C_VEL
LIN {X 0,Y 242.394,Z 522.133,A -85,B 0,C 180,E1 -19439.169,E2 -19439.169} C_VEL
LIN {X 0,Y 242.622,Z 525.353,A -85,B 0,C 180,E1 -19441.659,E2 -19441.659} C_VEL
LIN {X 0,Y 243.456,Z 528.485,A -85,B 0,C 180,E1 -19444.968,E2 -19444.968} C_VEL
LIN {X 0,Y 244.877,Z 530.34,A -85,B 0,C 180,E1 -19448.25,E2 -19448.25} C_VEL
LIN {X 0,Y 246.995,Z 530.937,A -85,B 0,C 180,E1 -19451.489,E2 -19451.489} C_VEL
LIN {X 0,Y 249.733,Z 530.332,A -85,B 0,C 180,E1 -19454.671,E2 -19454.671} C_VEL
LIN {X 0,Y 252.995,Z 528.574,A -85,B 0,C 180,E1 -19457.792,E2 -19457.792} C_VEL
LIN {X 0,Y 257.003,Z 525.587,A -85,B 0,C 180,E1 -19460.824,E2 -19460.824} C_VEL
LIN {X 0,Y 261.701,Z 521.35,A -85,B 0,C 180,E1 -19463.755,E2 -19463.755} C_VEL
LIN {X 0,Y 267.106,Z 515.78,A -85,B 0,C 180,E1 -19466.57,E2 -19466.57} C_VEL
LIN {X 0,Y 273.028,Z 508.91,A -85,B 0,C 180,E1 -19469.233,E2 -19469.233} C_VEL
LIN {X 0,Y 276.232,Z 504.475,A -85,B 0,C 180,E1 -19470.941,E2 -19470.941} C_VEL
LIN {X 0,Y 277.623,Z 502,A -85,B 0,C 180,E1 -19472.016,E2 -19472.016} C_VEL
LIN {X 0,Y 280.601,Z 495.865,A -85,B 0,C 180,E1 -19474.966,E2 -19474.966} C_VEL
LIN {X 0,Y 280.788,Z 495.503,A -85,B 0,C 180,E1 -19475.147,E2 -19475.147} C_VEL
LIN {X 0,Y 280.305,Z 494.589,A -85,B 0,C 180,E1 -19476.995,E2 -19476.995} C_VEL
LIN {X 0,Y 279.559,Z 494.607,A -85,B 0,C 180,E1 -19478.938,E2 -19478.938} C_VEL
LIN {X 0,Y 278.888,Z 495.437,A -85,B 0,C 180,E1 -19480.935,E2 -19480.935} C_VEL
LIN {X 0,Y 278.17,Z 497.376,A -85,B 0,C 180,E1 -19483.012,E2 -19483.012} C_VEL
LIN {X 0,Y 277.384,Z 499.253,A -85,B 0,C 180,E1 -19484.062,E2 -19484.062} C_VEL
LIN {X 0,Y 274.385,Z 506.071,A -85,B 0,C 180,E1 -19486.58,E2 -19486.58} C_VEL
LIN {X 0,Y 271.108,Z 514.416,A -85,B 0,C 180,E1 -19489.192,E2 -19489.192} C_VEL
LIN {X 0,Y 267.261,Z 523.982,A -85,B 0,C 180,E1 -19491.832,E2 -19491.832} C_VEL
LIN {X 0,Y 263.385,Z 532.567,A -85,B 0,C 180,E1 -19494.052,E2 -19494.052} C_VEL
LIN {X 0,Y 258.827,Z 541.079,A -85,B 0,C 180,E1 -19496.174,E2 -19496.174} C_VEL
LIN {X 0,Y 252.377,Z 552.604,A -85,B 0,C 180,E1 -19499.454,E2 -19499.454} C_VEL
LIN {X 0,Y 247.592,Z 559.913,A -85,B 0,C 180,E1 -19501.775,E2 -19501.775} C_VEL
LIN {X 0,Y 242.463,Z 568.476,A -85,B 0,C 180,E1 -19505.145,E2 -19505.145} C_VEL
LIN {X 0,Y 238.643,Z 575.114,A -85,B 0,C 180,E1 -19508.398,E2 -19508.398} C_VEL
LIN {X 0,Y 236.011,Z 580.567,A -85,B 0,C 180,E1 -19511.778,E2 -19511.778} C_VEL
LIN {X 0,Y 234.667,Z 583.902,A -85,B 0,C 180,E1 -19514.361,E2 -19514.361} C_VEL
LIN {X 0,Y 233.816,Z 587.372,A -85,B 0,C 180,E1 -19517.852,E2 -19517.852} C_VEL
LIN {X 0,Y 233.823,Z 589.652,A -85,B 0,C 180,E1 -19521.355,E2 -19521.355} C_VEL
LIN {X 0,Y 234.021,Z 590.078,A -85,B 0,C 180,E1 -19522.323,E2 -19522.323} C_VEL
LIN {X 0,Y 234.395,Z 592.128,A -85,B 0,C 180,E1 -19524.837,E2 -19524.837} C_VEL
LIN {X 0,Y 235.093,Z 593.457,A -85,B 0,C 180,E1 -19528.285,E2 -19528.285} C_VEL
LIN {X 0,Y 235.479,Z 593.502,A -85,B 0,C 180,E1 -19529.998,E2 -19529.998} C_VEL
LIN {X 0,Y 235.192,Z 593.02,A -85,B 0,C 180,E1 -19531.71,E2 -19531.71} C_VEL
LIN {X 0,Y 234.591,Z 590.684,A -85,B 0,C 180,E1 -19535.155,E2 -19535.155} C_VEL
LIN {X 0,Y 234.225,Z 587.393,A -85,B 0,C 180,E1 -19538.039,E2 -19538.039} C_VEL
LIN {X 0,Y 234.104,Z 583.754,A -85,B 0,C 180,E1 -19540.375,E2 -19540.375} C_VEL
LIN {X 0,Y 234.392,Z 577.609,A -85,B 0,C 180,E1 -19543.435,E2 -19543.435} C_VEL
LIN {X 0,Y 235.176,Z 570.853,A -85,B 0,C 180,E1 -19546.045,E2 -19546.045} C_VEL
LIN {X 0,Y 236.375,Z 562.49,A -85,B 0,C 180,E1 -19548.638,E2 -19548.638} C_VEL
LIN {X 0,Y 237.904,Z 553.994,A -85,B 0,C 180,E1 -19550.76,E2 -19550.76} C_VEL
LIN {X 0,Y 239.621,Z 543.515,A -85,B 0,C 180,E1 -19552.866,E2 -19552.866} C_VEL
LIN {X 0,Y 240.778,Z 535.988,A -85,B 0,C 180,E1 -19554.117,E2 -19554.117} C_VEL
LIN {X 0,Y 240.411,Z 524.388,A -85,B 0,C 180,E1 -19555.851,E2 -19555.851} C_VEL
LIN {X 0,Y 239.677,Z 510.824,A -85,B 0,C 180,E1 -19557.477,E2 -19557.477} C_VEL
LIN {X 0,Y 238.862,Z 497.997,A -85,B 0,C 180,E1 -19558.647,E2 -19558.647} C_VEL
LIN {X 0,Y 237.736,Z 484.73,A -85,B 0,C 180,E1 -19559.516,E2 -19559.516} C_VEL
LIN {X 0,Y 236.438,Z 470.808,A -85,B 0,C 180,E1 -19560.186,E2 -19560.186} C_VEL
LIN {X 0,Y 236.079,Z 462.446,A -85,B 0,C 180,E1 -19561.295,E2 -19561.295} C_VEL
LIN {X 0,Y 237.695,Z 453.306,A -85,B 0,C 180,E1 -19566.25,E2 -19566.25} C_VEL
LIN {X 0,Y 239.259,Z 445.917,A -85,B 0,C 180,E1 -19570.255,E2 -19570.255} C_VEL
LIN {X 0,Y 239.634,Z 443.023,A -85,B 0,C 180,E1 -19571.849,E2 -19571.849} C_VEL
LIN {X 0,Y 238.121,Z 435.707,A -85,B 0,C 180,E1 -19576.085,E2 -19576.085} C_VEL
LIN {X 0,Y 236.608,Z 428.342,A -85,B 0,C 180,E1 -19580.556,E2 -19580.556} C_VEL
LIN {X 0,Y 235.397,Z 422.093,A -85,B 0,C 180,E1 -19584.509,E2 -19584.509} C_VEL
LIN {X 0,Y 234.965,Z 419.842,A -85,B 0,C 180,E1 -19585.999,E2 -19585.999} C_VEL
LIN {X 0,Y 234.961,Z 419.838,A -85,B 0,C 180,E1 -19590.156,E2 -19590.156} C_VEL
LIN {X 0,Y 234.986,Z 419.837,A -85,B 0,C 180,E1 -19593.793,E2 -19593.793} C_VEL
LIN {X 0,Y 235.002,Z 419.834,A -85,B 0,C 180,E1 -19598.969,E2 -19598.969} C_VEL
LIN {X 0,Y 235.087,Z 419.826,A -85,B 0,C 180,E1 -19603.059,E2 -19603.059} C_VEL
LIN {X 0,Y 235.138,Z 419.819,A -85,B 0,C 180,E1 -19607.924,E2 -19607.924} C_VEL
LIN {X 0,Y 235.367,Z 419.791,A -85,B 0,C 180,E1 -19611.414,E2 -19611.414} C_VEL
LIN {X 0,Y 235.395,Z 419.788,A -85,B 0,C 180,E1 -19613.142,E2 -19613.142} C_VEL
LIN {X 0,Y 235.59,Z 419.764,A -85,B 0,C 180,E1 -19618.291,E2 -19618.291} C_VEL
LIN {X 0,Y 235.59,Z 419.76,A -85,B 0,C 180,E1 -19621.71,E2 -19621.71} C_VEL
LIN {X 0,Y 235.396,Z 419.772,A -85,B 0,C 180,E1 -19626.859,E2 -19626.859} C_VEL
LIN {X 0,Y 235.229,Z 419.787,A -85,B 0,C 180,E1 -19630.327,E2 -19630.327} C_VEL
LIN {X 0,Y 235.106,Z 419.822,A -85,B 0,C 180,E1 -19635.607,E2 -19635.607} C_VEL
LIN {X 0,Y 235.001,Z 419.837,A -85,B 0,C 180,E1 -19639.207,E2 -19639.207} C_VEL
LIN {X 0,Y 234.953,Z 419.839,A -85,B 0,C 180,E1 -19642.884,E2 -19642.884} C_VEL
LIN {X 0,Y 234.961,Z 419.836,A -85,B 0,C 180,E1 -19646.659,E2 -19646.659} C_VEL
LIN {X 0,Y 234.916,Z 419.822,A -85,B 0,C 180,E1 -19650.571,E2 -19650.571} C_VEL
LIN {X 0,Y 234.924,Z 419.846,A -85,B 0,C 180,E1 -19654.64,E2 -19654.64} C_VEL
LIN {X 0,Y 234.936,Z 419.827,A -85,B 0,C 180,E1 -19658.946,E2 -19658.946} C_VEL
LIN {X 0,Y 234.886,Z 419.847,A -85,B 0,C 180,E1 -19663.487,E2 -19663.487} C_VEL
LIN {X 0,Y 234.925,Z 419.837,A -85,B 0,C 180,E1 -19666.526,E2 -19666.526} C_VEL
LIN {X 0,Y 234.952,Z 419.834,A -85,B 0,C 180,E1 -19671.088,E2 -19671.088} C_VEL
LIN {X 0,Y 234.958,Z 419.842,A -85,B 0,C 180,E1 -19675.369,E2 -19675.369} C_VEL
LIN {X 0,Y 234.968,Z 419.837,A -85,B 0,C 180,E1 -19680.159,E2 -19680.159} C_VEL
LIN {X 0,Y 234.985,Z 419.835,A -85,B 0,C 180,E1 -19682.739,E2 -19682.739} C_VEL
LIN {X 0,Y 235.993,Z 422.669,A -85,B 0,C 180,E1 -19683,E2 -19683} C_VEL
LIN {X 0,Y 241.384,Z 433.326,A -85,B 0,C 180,E1 -19684.284,E2 -19684.284} C_VEL
LIN {X 0,Y 245.699,Z 444.122,A -85,B 0,C 180,E1 -19685.69,E2 -19685.69} C_VEL
LIN {X 0,Y 249.076,Z 454.583,A -85,B 0,C 180,E1 -19687.211,E2 -19687.211} C_VEL
LIN {X 0,Y 249.157,Z 457.23,A -85,B 0,C 180,E1 -19687.538,E2 -19687.538} C_VEL
LIN {X 0,Y 247.64,Z 468.671,A -85,B 0,C 180,E1 -19689.007,E2 -19689.007} C_VEL
LIN {X 0,Y 245.941,Z 478.61,A -85,B 0,C 180,E1 -19690.603,E2 -19690.603} C_VEL
LIN {X 0,Y 244.232,Z 487.705,A -85,B 0,C 180,E1 -19692.415,E2 -19692.415} C_VEL
LIN {X 0,Y 242.338,Z 496.052,A -85,B 0,C 180,E1 -19694.441,E2 -19694.441} C_VEL
LIN {X 0,Y 240.526,Z 504.11,A -85,B 0,C 180,E1 -19696.914,E2 -19696.914} C_VEL
LIN {X 0,Y 239.158,Z 509.634,A -85,B 0,C 180,E1 -19698.99,E2 -19698.99} C_VEL
LIN {X 0,Y 237.973,Z 514.981,A -85,B 0,C 180,E1 -19701.51,E2 -19701.51} C_VEL
LIN {X 0,Y 236.864,Z 519.196,A -85,B 0,C 180,E1 -19704.041,E2 -19704.041} C_VEL
LIN {X 0,Y 236.014,Z 522.373,A -85,B 0,C 180,E1 -19706.588,E2 -19706.588} C_VEL
LIN {X 0,Y 235.562,Z 525.115,A -85,B 0,C 180,E1 -19710.002,E2 -19710.002} C_VEL
LIN {X 0,Y 235.555,Z 525.866,A -85,B 0,C 180,E1 -19711.712,E2 -19711.712} C_VEL
LIN {X 0,Y 235.419,Z 526.282,A -85,B 0,C 180,E1 -19715.14,E2 -19715.14} C_VEL
LIN {X 0,Y 235.785,Z 525.894,A -85,B 0,C 180,E1 -19716.849,E2 -19716.849} C_VEL
LIN {X 0,Y 237.067,Z 523.849,A -85,B 0,C 180,E1 -19720.248,E2 -19720.248} C_VEL
LIN {X 0,Y 238.261,Z 520.764,A -85,B 0,C 180,E1 -19723.242,E2 -19723.242} C_VEL
LIN {X 0,Y 239.837,Z 516.339,A -85,B 0,C 180,E1 -19726.165,E2 -19726.165} C_VEL
LIN {X 0,Y 241.465,Z 511.28,A -85,B 0,C 180,E1 -19728.674,E2 -19728.674} C_VEL
LIN {X 0,Y 243.367,Z 504.898,A -85,B 0,C 180,E1 -19731.162,E2 -19731.162} C_VEL
LIN {X 0,Y 245.718,Z 496.912,A -85,B 0,C 180,E1 -19733.607,E2 -19733.607} C_VEL
LIN {X 0,Y 247.92,Z 488.656,A -85,B 0,C 180,E1 -19735.616,E2 -19735.616} C_VEL
LIN {X 0,Y 250.197,Z 478.466,A -85,B 0,C 180,E1 -19737.614,E2 -19737.614} C_VEL
LIN {X 0,Y 252.089,Z 468.04,A -85,B 0,C 180,E1 -19739.257,E2 -19739.257} C_VEL
LIN {X 0,Y 253.02,Z 460.935,A -85,B 0,C 180,E1 -19740.193,E2 -19740.193} C_VEL
LIN {X 0,Y 250.367,Z 452.312,A -85,B 0,C 180,E1 -19741.684,E2 -19741.684} C_VEL
LIN {X 0,Y 246.441,Z 442.476,A -85,B 0,C 180,E1 -19743.285,E2 -19743.285} C_VEL
LIN {X 0,Y 240.959,Z 431.064,A -85,B 0,C 180,E1 -19745.012,E2 -19745.012} C_VEL
LIN {X 0,Y 236.63,Z 423.621,A -85,B 0,C 180,E1 -19746.118,E2 -19746.118} C_VEL
LIN {X 0,Y 235.134,Z 420.848,A -85,B 0,C 180,E1 -19746.484,E2 -19746.484} C_VEL
LIN {X 0,Y 235.019,Z 420.394,A -85,B 0,C 180,E1 -19746.543,E2 -19746.543} C_VEL
LIN {X 0,Y 234.923,Z 419.834,A -85,B 0,C 180,E1 -19746.886,E2 -19746.886} C_VEL
LIN {X 0,Y 234.948,Z 419.824,A -85,B 0,C 180,E1 -19748.945,E2 -19748.945} C_VEL
LIN {X 0,Y 234.891,Z 419.85,A -85,B 0,C 180,E1 -19753.487,E2 -19753.487} C_VEL
LIN {X 0,Y 234.887,Z 419.847,A -85,B 0,C 180,E1 -19756.513,E2 -19756.513} C_VEL
LIN {X 0,Y 234.924,Z 419.804,A -85,B 0,C 180,E1 -19761.079,E2 -19761.079} C_VEL
LIN {X 0,Y 234.936,Z 419.846,A -85,B 0,C 180,E1 -19765.362,E2 -19765.362} C_VEL
LIN {X 0,Y 234.928,Z 419.792,A -85,B 0,C 180,E1 -19769.431,E2 -19769.431} C_VEL
LIN {X 0,Y 235.034,Z 419.998,A -85,B 0,C 180,E1 -19773.396,E2 -19773.396} C_VEL
LIN {X 0,Y 238.728,Z 433.628,A -85,B 0,C 180,E1 -19775.132,E2 -19775.132} C_VEL
LIN {X 0,Y 242.464,Z 447.308,A -85,B 0,C 180,E1 -19777.19,E2 -19777.19} C_VEL
LIN {X 0,Y 242.978,Z 450.637,A -85,B 0,C 180,E1 -19777.711,E2 -19777.711} C_VEL
LIN {X 0,Y 241.443,Z 462.12,A -85,B 0,C 180,E1 -19779.555,E2 -19779.555} C_VEL
LIN {X 0,Y 239.916,Z 473.115,A -85,B 0,C 180,E1 -19781.644,E2 -19781.644} C_VEL
LIN {X 0,Y 238.475,Z 484.271,A -85,B 0,C 180,E1 -19784.18,E2 -19784.18} C_VEL
LIN {X 0,Y 237.095,Z 495.136,A -85,B 0,C 180,E1 -19787.154,E2 -19787.154} C_VEL
LIN {X 0,Y 236.148,Z 504.178,A -85,B 0,C 180,E1 -19790.146,E2 -19790.146} C_VEL
LIN {X 0,Y 235.411,Z 511.629,A -85,B 0,C 180,E1 -19793.141,E2 -19793.141} C_VEL
LIN {X 0,Y 235.029,Z 518.509,A -85,B 0,C 180,E1 -19796.571,E2 -19796.571} C_VEL
LIN {X 0,Y 235.333,Z 522.68,A -85,B 0,C 180,E1 -19799.144,E2 -19799.144} C_VEL
LIN {X 0,Y 235.558,Z 526.028,A -85,B 0,C 180,E1 -19801.709,E2 -19801.709} C_VEL
LIN {X 0,Y 236.461,Z 529.384,A -85,B 0,C 180,E1 -19805.115,E2 -19805.115} C_VEL
LIN {X 0,Y 237.946,Z 531.486,A -85,B 0,C 180,E1 -19808.492,E2 -19808.492} C_VEL
LIN {X 0,Y 240.192,Z 532.34,A -85,B 0,C 180,E1 -19811.819,E2 -19811.819} C_VEL
LIN {X 0,Y 243.083,Z 532.003,A -85,B 0,C 180,E1 -19815.082,E2 -19815.082} C_VEL
LIN {X 0,Y 246.517,Z 530.533,A -85,B 0,C 180,E1 -19818.276,E2 -19818.276} C_VEL
LIN {X 0,Y 250.743,Z 527.858,A -85,B 0,C 180,E1 -19821.369,E2 -19821.369} C_VEL
LIN {X 0,Y 255.658,Z 523.973,A -85,B 0,C 180,E1 -19824.352,E2 -19824.352} C_VEL
LIN {X 0,Y 261.292,Z 518.774,A -85,B 0,C 180,E1 -19827.21,E2 -19827.21} C_VEL
LIN {X 0,Y 268.063,Z 511.66,A -85,B 0,C 180,E1 -19830.134,E2 -19830.134} C_VEL
LIN {X 0,Y 275.352,Z 503.08,A -85,B 0,C 180,E1 -19832.845,E2 -19832.845} C_VEL
LIN {X 0,Y 280.018,Z 497.032,A -85,B 0,C 180,E1 -19834.382,E2 -19834.382} C_VEL
LIN {X 0,Y 280.601,Z 495.865,A -85,B 0,C 180,E1 -19834.966,E2 -19834.966} C_VEL
LIN {X 0,Y 280.852,Z 494.985,A -85,B 0,C 180,E1 -19835.715,E2 -19835.715} C_VEL
LIN {X 0,Y 280.393,Z 494.962,A -85,B 0,C 180,E1 -19836.492,E2 -19836.492} C_VEL
LIN {X 0,Y 278.894,Z 496.019,A -85,B 0,C 180,E1 -19837.649,E2 -19837.649} C_VEL
LIN {X 0,Y 274.529,Z 500.492,A -85,B 0,C 180,E1 -19840.433,E2 -19840.433} C_VEL
LIN {X 0,Y 273.955,Z 501.352,A -85,B 0,C 180,E1 -19841.293,E2 -19841.293} C_VEL
LIN {X 0,Y 273.796,Z 501.763,A -85,B 0,C 180,E1 -19841.891,E2 -19841.891} C_VEL
LIN {X 0,Y 273.313,Z 502.977,A -85,B 0,C 180,E1 -19842.919,E2 -19842.919} C_VEL
LIN {X 0,Y 271.791,Z 505.905,A -85,B 0,C 180,E1 -19844.28,E2 -19844.28} C_VEL
LIN {X 0,Y 268.076,Z 513.536,A -85,B 0,C 180,E1 -19847.027,E2 -19847.027} C_VEL
LIN {X 0,Y 264.583,Z 521.131,A -85,B 0,C 180,E1 -19849.398,E2 -19849.398} C_VEL
LIN {X 0,Y 260.755,Z 529.122,A -85,B 0,C 180,E1 -19851.689,E2 -19851.689} C_VEL
LIN {X 0,Y 255.606,Z 538.608,A -85,B 0,C 180,E1 -19854.246,E2 -19854.246} C_VEL
LIN {X 0,Y 248.463,Z 550.02,A -85,B 0,C 180,E1 -19857.489,E2 -19857.489} C_VEL
LIN {X 0,Y 244.746,Z 555.738,A -85,B 0,C 180,E1 -19859.354,E2 -19859.354} C_VEL
LIN {X 0,Y 240.43,Z 561.876,A -85,B 0,C 180,E1 -19861.553,E2 -19861.553} C_VEL
LIN {X 0,Y 234.911,Z 570.221,A -85,B 0,C 180,E1 -19865.236,E2 -19865.236} C_VEL
LIN {X 0,Y 231.186,Z 576.226,A -85,B 0,C 180,E1 -19868.603,E2 -19868.603} C_VEL
LIN {X 0,Y 228.396,Z 581.649,A -85,B 0,C 180,E1 -19872.535,E2 -19872.535} C_VEL
LIN {X 0,Y 227.142,Z 584.867,A -85,B 0,C 180,E1 -19875.667,E2 -19875.667} C_VEL
LIN {X 0,Y 226.695,Z 587.524,A -85,B 0,C 180,E1 -19879.278,E2 -19879.278} C_VEL
LIN {X 0,Y 226.943,Z 589.273,A -85,B 0,C 180,E1 -19882.297,E2 -19882.297} C_VEL
LIN {X 0,Y 227.314,Z 591.134,A -85,B 0,C 180,E1 -19884.676,E2 -19884.676} C_VEL
LIN {X 0,Y 228.019,Z 592.449,A -85,B 0,C 180,E1 -19888.232,E2 -19888.232} C_VEL
LIN {X 0,Y 228.443,Z 592.493,A -85,B 0,C 180,E1 -19889.998,E2 -19889.998} C_VEL
LIN {X 0,Y 228.121,Z 591.991,A -85,B 0,C 180,E1 -19891.764,E2 -19891.764} C_VEL
LIN {X 0,Y 227.733,Z 591.014,A -85,B 0,C 180,E1 -19893.537,E2 -19893.537} C_VEL
LIN {X 0,Y 227.505,Z 589.633,A -85,B 0,C 180,E1 -19895.316,E2 -19895.316} C_VEL
LIN {X 0,Y 227.149,Z 586.59,A -85,B 0,C 180,E1 -19898.077,E2 -19898.077} C_VEL
LIN {X 0,Y 227.024,Z 582.657,A -85,B 0,C 180,E1 -19900.702,E2 -19900.702} C_VEL
LIN {X 0,Y 227.383,Z 576.483,A -85,B 0,C 180,E1 -19903.857,E2 -19903.857} C_VEL
LIN {X 0,Y 228.359,Z 568.728,A -85,B 0,C 180,E1 -19906.889,E2 -19906.889} C_VEL
LIN {X 0,Y 229.568,Z 561.319,A -85,B 0,C 180,E1 -19909.212,E2 -19909.212} C_VEL
LIN {X 0,Y 231.178,Z 552.797,A -85,B 0,C 180,E1 -19911.394,E2 -19911.394} C_VEL
LIN {X 0,Y 232.806,Z 543.456,A -85,B 0,C 180,E1 -19913.34,E2 -19913.34} C_VEL
LIN {X 0,Y 233.912,Z 536.006,A -85,B 0,C 180,E1 -19914.636,E2 -19914.636} C_VEL
LIN {X 0,Y 233.651,Z 524.704,A -85,B 0,C 180,E1 -19916.424,E2 -19916.424} C_VEL
LIN {X 0,Y 233.108,Z 512.742,A -85,B 0,C 180,E1 -19917.959,E2 -19917.959} C_VEL
LIN {X 0,Y 232.429,Z 499.317,A -85,B 0,C 180,E1 -19919.289,E2 -19919.289} C_VEL
LIN {X 0,Y 231.445,Z 485.83,A -85,B 0,C 180,E1 -19920.264,E2 -19920.264} C_VEL
LIN {X 0,Y 229.887,Z 469.454,A -85,B 0,C 180,E1 -19921.13,E2 -19921.13} C_VEL
LIN {X 0,Y 229.312,Z 460.321,A -85,B 0,C 180,E1 -19922.432,E2 -19922.432} C_VEL
LIN {X 0,Y 230.655,Z 453.173,A -85,B 0,C 180,E1 -19926.45,E2 -19926.45} C_VEL
LIN {X 0,Y 232.342,Z 445.33,A -85,B 0,C 180,E1 -19930.869,E2 -19930.869} C_VEL
LIN {X 0,Y 232.567,Z 443.919,A -85,B 0,C 180,E1 -19931.666,E2 -19931.666} C_VEL
LIN {X 0,Y 231.236,Z 437.207,A -85,B 0,C 180,E1 -19935.65,E2 -19935.65} C_VEL
LIN {X 0,Y 229.437,Z 428.461,A -85,B 0,C 180,E1 -19941.102,E2 -19941.102} C_VEL
LIN {X 0,Y 227.973,Z 421.007,A -85,B 0,C 180,E1 -19946.03,E2 -19946.03} C_VEL
LIN {X 0,Y 227.918,Z 420.719,A -85,B 0,C 180,E1 -19946.359,E2 -19946.359} C_VEL
LIN {X 0,Y 227.911,Z 420.716,A -85,B 0,C 180,E1 -19950.437,E2 -19950.437} C_VEL
LIN {X 0,Y 227.92,Z 420.717,A -85,B 0,C 180,E1 -19954.425,E2 -19954.425} C_VEL
LIN {X 0,Y 227.953,Z 420.714,A -85,B 0,C 180,E1 -19958.287,E2 -19958.287} C_VEL
LIN {X 0,Y 228.026,Z 420.708,A -85,B 0,C 180,E1 -19962.825,E2 -19962.825} C_VEL
LIN {X 0,Y 228.085,Z 420.698,A -85,B 0,C 180,E1 -19967.544,E2 -19967.544} C_VEL
LIN {X 0,Y 228.297,Z 420.669,A -85,B 0,C 180,E1 -19971.146,E2 -19971.146} C_VEL
LIN {X 0,Y 228.346,Z 420.668,A -85,B 0,C 180,E1 -19972.929,E2 -19972.929} C_VEL
LIN {X 0,Y 228.548,Z 420.641,A -85,B 0,C 180,E1 -19978.238,E2 -19978.238} C_VEL
LIN {X 0,Y 228.549,Z 420.638,A -85,B 0,C 180,E1 -19981.763,E2 -19981.763} C_VEL
LIN {X 0,Y 228.347,Z 420.648,A -85,B 0,C 180,E1 -19987.072,E2 -19987.072} C_VEL
LIN {X 0,Y 228.155,Z 420.669,A -85,B 0,C 180,E1 -19990.651,E2 -19990.651} C_VEL
LIN {X 0,Y 228.057,Z 420.702,A -85,B 0,C 180,E1 -19994.273,E2 -19994.273} C_VEL
LIN {X 0,Y 227.995,Z 420.705,A -85,B 0,C 180,E1 -19997.954,E2 -19997.954} C_VEL
LIN {X 0,Y 227.922,Z 420.713,A -85,B 0,C 180,E1 -20002.331,E2 -20002.331} C_VEL
LIN {X 0,Y 227.935,Z 420.711,A -85,B 0,C 180,E1 -20006.604,E2 -20006.604} C_VEL
LIN {X 0,Y 227.89,Z 420.694,A -85,B 0,C 180,E1 -20010.293,E2 -20010.293} C_VEL
LIN {X 0,Y 227.871,Z 420.723,A -85,B 0,C 180,E1 -20013.722,E2 -20013.722} C_VEL
LIN {X 0,Y 227.838,Z 420.708,A -85,B 0,C 180,E1 -20018.093,E2 -20018.093} C_VEL
LIN {X 0,Y 227.808,Z 420.731,A -85,B 0,C 180,E1 -20022.744,E2 -20022.744} C_VEL
LIN {X 0,Y 227.865,Z 420.725,A -85,B 0,C 180,E1 -20027.273,E2 -20027.273} C_VEL
LIN {X 0,Y 227.868,Z 420.72,A -85,B 0,C 180,E1 -20031.917,E2 -20031.917} C_VEL
LIN {X 0,Y 227.888,Z 420.722,A -85,B 0,C 180,E1 -20036.375,E2 -20036.375} C_VEL
LIN {X 0,Y 227.902,Z 420.722,A -85,B 0,C 180,E1 -20041.205,E2 -20041.205} C_VEL
LIN {X 0,Y 227.962,Z 420.913,A -85,B 0,C 180,E1 -20041.78,E2 -20041.78} C_VEL
LIN {X 0,Y 229.022,Z 423.673,A -85,B 0,C 180,E1 -20042.042,E2 -20042.042} C_VEL
LIN {X 0,Y 234.907,Z 435.219,A -85,B 0,C 180,E1 -20043.528,E2 -20043.528} C_VEL
LIN {X 0,Y 239.204,Z 445.995,A -85,B 0,C 180,E1 -20045.014,E2 -20045.014} C_VEL
LIN {X 0,Y 242.592,Z 456.232,A -85,B 0,C 180,E1 -20046.592,E2 -20046.592} C_VEL
LIN {X 0,Y 242.705,Z 458.764,A -85,B 0,C 180,E1 -20046.926,E2 -20046.926} C_VEL
LIN {X 0,Y 241.128,Z 469.977,A -85,B 0,C 180,E1 -20048.412,E2 -20048.412} C_VEL
LIN {X 0,Y 239.383,Z 479.719,A -85,B 0,C 180,E1 -20050.02,E2 -20050.02} C_VEL
LIN {X 0,Y 237.57,Z 488.919,A -85,B 0,C 180,E1 -20051.906,E2 -20051.906} C_VEL
LIN {X 0,Y 235.607,Z 497.226,A -85,B 0,C 180,E1 -20053.985,E2 -20053.985} C_VEL
LIN {X 0,Y 233.704,Z 505.248,A -85,B 0,C 180,E1 -20056.525,E2 -20056.525} C_VEL
LIN {X 0,Y 232.293,Z 510.746,A -85,B 0,C 180,E1 -20058.661,E2 -20058.661} C_VEL
LIN {X 0,Y 231.036,Z 516.073,A -85,B 0,C 180,E1 -20061.253,E2 -20061.253} C_VEL
LIN {X 0,Y 229.88,Z 520.269,A -85,B 0,C 180,E1 -20063.859,E2 -20063.859} C_VEL
LIN {X 0,Y 229.003,Z 523.427,A -85,B 0,C 180,E1 -20066.483,E2 -20066.483} C_VEL
LIN {X 0,Y 228.535,Z 526.149,A -85,B 0,C 180,E1 -20070.002,E2 -20070.002} C_VEL
LIN {X 0,Y 228.53,Z 526.884,A -85,B 0,C 180,E1 -20071.764,E2 -20071.764} C_VEL
LIN {X 0,Y 228.413,Z 527.282,A -85,B 0,C 180,E1 -20075.298,E2 -20075.298} C_VEL
LIN {X 0,Y 228.802,Z 526.881,A -85,B 0,C 180,E1 -20077.059,E2 -20077.059} C_VEL
LIN {X 0,Y 230.15,Z 524.812,A -85,B 0,C 180,E1 -20080.559,E2 -20080.559} C_VEL
LIN {X 0,Y 231.424,Z 521.708,A -85,B 0,C 180,E1 -20083.638,E2 -20083.638} C_VEL
LIN {X 0,Y 233.088,Z 517.251,A -85,B 0,C 180,E1 -20086.647,E2 -20086.647} C_VEL
LIN {X 0,Y 234.794,Z 512.17,A -85,B 0,C 180,E1 -20089.226,E2 -20089.226} C_VEL
LIN {X 0,Y 236.789,Z 505.763,A -85,B 0,C 180,E1 -20091.779,E2 -20091.779} C_VEL
LIN {X 0,Y 239.276,Z 497.74,A -85,B 0,C 180,E1 -20094.282,E2 -20094.282} C_VEL
LIN {X 0,Y 241.57,Z 489.434,A -85,B 0,C 180,E1 -20096.34,E2 -20096.34} C_VEL
LIN {X 0,Y 243.962,Z 479.195,A -85,B 0,C 180,E1 -20098.382,E2 -20098.382} C_VEL
LIN {X 0,Y 246.039,Z 468.268,A -85,B 0,C 180,E1 -20100.122,E2 -20100.122} C_VEL
LIN {X 0,Y 246.704,Z 462.953,A -85,B 0,C 180,E1 -20100.851,E2 -20100.851} C_VEL
LIN {X 0,Y 243.38,Z 452.35,A -85,B 0,C 180,E1 -20102.764,E2 -20102.764} C_VEL
LIN {X 0,Y 238.438,Z 440.702,A -85,B 0,C 180,E1 -20104.752,E2 -20104.752} C_VEL
LIN {X 0,Y 233.674,Z 431.412,A -85,B 0,C 180,E1 -20106.247,E2 -20106.247} C_VEL
LIN {X 0,Y 229.736,Z 424.661,A -85,B 0,C 180,E1 -20107.307,E2 -20107.307} C_VEL
LIN {X 0,Y 228.262,Z 422.145,A -85,B 0,C 180,E1 -20107.684,E2 -20107.684} C_VEL
LIN {X 0,Y 228.046,Z 421.423,A -85,B 0,C 180,E1 -20107.804,E2 -20107.804} C_VEL
LIN {X 0,Y 227.897,Z 420.7,A -85,B 0,C 180,E1 -20108.215,E2 -20108.215} C_VEL
LIN {X 0,Y 227.816,Z 420.727,A -85,B 0,C 180,E1 -20112.743,E2 -20112.743} C_VEL
LIN {X 0,Y 227.813,Z 420.733,A -85,B 0,C 180,E1 -20117.257,E2 -20117.257} C_VEL
LIN {X 0,Y 227.85,Z 420.686,A -85,B 0,C 180,E1 -20121.909,E2 -20121.909} C_VEL
LIN {X 0,Y 227.886,Z 420.72,A -85,B 0,C 180,E1 -20126.378,E2 -20126.378} C_VEL
LIN {X 0,Y 227.911,Z 420.661,A -85,B 0,C 180,E1 -20130.436,E2 -20130.436} C_VEL
LIN {X 0,Y 227.996,Z 420.859,A -85,B 0,C 180,E1 -20133.037,E2 -20133.037} C_VEL
LIN {X 0,Y 231.752,Z 434.9,A -85,B 0,C 180,E1 -20134.877,E2 -20134.877} C_VEL
LIN {X 0,Y 235.49,Z 448.723,A -85,B 0,C 180,E1 -20137.02,E2 -20137.02} C_VEL
LIN {X 0,Y 235.983,Z 451.089,A -85,B 0,C 180,E1 -20137.407,E2 -20137.407} C_VEL
LIN {X 0,Y 234.553,Z 461.76,A -85,B 0,C 180,E1 -20139.156,E2 -20139.156} C_VEL
LIN {X 0,Y 232.802,Z 473.98,A -85,B 0,C 180,E1 -20141.519,E2 -20141.519} C_VEL
LIN {X 0,Y 231.364,Z 485.167,A -85,B 0,C 180,E1 -20144.134,E2 -20144.134} C_VEL
LIN {X 0,Y 229.969,Z 496.054,A -85,B 0,C 180,E1 -20147.199,E2 -20147.199} C_VEL
LIN {X 0,Y 229.017,Z 505.123,A -85,B 0,C 180,E1 -20150.282,E2 -20150.282} C_VEL
LIN {X 0,Y 228.356,Z 511.611,A -85,B 0,C 180,E1 -20152.928,E2 -20152.928} C_VEL
LIN {X 0,Y 227.962,Z 518.807,A -85,B 0,C 180,E1 -20156.464,E2 -20156.464} C_VEL
LIN {X 0,Y 228.246,Z 523.106,A -85,B 0,C 180,E1 -20159.117,E2 -20159.117} C_VEL
LIN {X 0,Y 228.492,Z 526.682,A -85,B 0,C 180,E1 -20161.762,E2 -20161.762} C_VEL
LIN {X 0,Y 229.467,Z 530.259,A -85,B 0,C 180,E1 -20165.271,E2 -20165.271} C_VEL
LIN {X 0,Y 231.017,Z 532.603,A -85,B 0,C 180,E1 -20168.749,E2 -20168.749} C_VEL
LIN {X 0,Y 233.39,Z 533.709,A -85,B 0,C 180,E1 -20172.168,E2 -20172.168} C_VEL
LIN {X 0,Y 236.435,Z 533.635,A -85,B 0,C 180,E1 -20175.517,E2 -20175.517} C_VEL
LIN {X 0,Y 240.04,Z 532.449,A -85,B 0,C 180,E1 -20178.787,E2 -20178.787} C_VEL
LIN {X 0,Y 244.478,Z 530.074,A -85,B 0,C 180,E1 -20181.944,E2 -20181.944} C_VEL
LIN {X 0,Y 249.627,Z 526.524,A -85,B 0,C 180,E1 -20184.98,E2 -20184.98} C_VEL
LIN {X 0,Y 255.532,Z 521.728,A -85,B 0,C 180,E1 -20187.876,E2 -20187.876} C_VEL
LIN {X 0,Y 262.096,Z 515.628,A -85,B 0,C 180,E1 -20190.629,E2 -20190.629} C_VEL
LIN {X 0,Y 269.222,Z 508.126,A -85,B 0,C 180,E1 -20193.243,E2 -20193.243} C_VEL
LIN {X 0,Y 275.534,Z 500.777,A -85,B 0,C 180,E1 -20195.29,E2 -20195.29} C_VEL
LIN {X 0,Y 275.697,Z 500.197,A -85,B 0,C 180,E1 -20195.895,E2 -20195.895} C_VEL
LIN {X 0,Y 275.2,Z 499.829,A -85,B 0,C 180,E1 -20197.8,E2 -20197.8} C_VEL
LIN {X 0,Y 274.495,Z 500.327,A -85,B 0,C 180,E1 -20199.815,E2 -20199.815} C_VEL
LIN {X 0,Y 273.955,Z 501.352,A -85,B 0,C 180,E1 -20201.293,E2 -20201.293} C_VEL
LIN {X 0,Y 273.379,Z 502.356,A -85,B 0,C 180,E1 -20202.072,E2 -20202.072} C_VEL
LIN {X 0,Y 272.298,Z 504.022,A -85,B 0,C 180,E1 -20202.782,E2 -20202.782} C_VEL
LIN {X 0,Y 270.867,Z 506.126,A -85,B 0,C 180,E1 -20203.435,E2 -20203.435} C_VEL
LIN {X 0,Y 263.323,Z 517.013,A -85,B 0,C 180,E1 -20206.212,E2 -20206.212} C_VEL
LIN {X 0,Y 262.694,Z 518.097,A -85,B 0,C 180,E1 -20206.569,E2 -20206.569} C_VEL
LIN {X 0,Y 258.3,Z 526.294,A -85,B 0,C 180,E1 -20209.229,E2 -20209.229} C_VEL
LIN {X 0,Y 253.86,Z 534.15,A -85,B 0,C 180,E1 -20211.569,E2 -20211.569} C_VEL
LIN {X 0,Y 249.175,Z 541.554,A -85,B 0,C 180,E1 -20213.678,E2 -20213.678} C_VEL
LIN {X 0,Y 242.567,Z 551.06,A -85,B 0,C 180,E1 -20216.597,E2 -20216.597} C_VEL
LIN {X 0,Y 238.715,Z 556.498,A -85,B 0,C 180,E1 -20218.493,E2 -20218.493} C_VEL
LIN {X 0,Y 233.391,Z 563.355,A -85,B 0,C 180,E1 -20221.195,E2 -20221.195} C_VEL
LIN {X 0,Y 227.346,Z 571.692,A -85,B 0,C 180,E1 -20225.332,E2 -20225.332} C_VEL
LIN {X 0,Y 223.749,Z 577.081,A -85,B 0,C 180,E1 -20228.823,E2 -20228.823} C_VEL
LIN {X 0,Y 220.882,Z 582.335,A -85,B 0,C 180,E1 -20233.358,E2 -20233.358} C_VEL
LIN {X 0,Y 219.799,Z 585.324,A -85,B 0,C 180,E1 -20237.064,E2 -20237.064} C_VEL
LIN {X 0,Y 219.742,Z 587.171,A -85,B 0,C 180,E1 -20240.796,E2 -20240.796} C_VEL
LIN {X 0,Y 220.236,Z 590.139,A -85,B 0,C 180,E1 -20244.505,E2 -20244.505} C_VEL
LIN {X 0,Y 220.945,Z 591.441,A -85,B 0,C 180,E1 -20248.175,E2 -20248.175} C_VEL
LIN {X 0,Y 221.405,Z 591.483,A -85,B 0,C 180,E1 -20249.998,E2 -20249.998} C_VEL
LIN {X 0,Y 221.049,Z 590.961,A -85,B 0,C 180,E1 -20251.82,E2 -20251.82} C_VEL
LIN {X 0,Y 220.659,Z 589.974,A -85,B 0,C 180,E1 -20253.65,E2 -20253.65} C_VEL
LIN {X 0,Y 220.421,Z 588.581,A -85,B 0,C 180,E1 -20255.487,E2 -20255.487} C_VEL
LIN {X 0,Y 220.085,Z 585.759,A -85,B 0,C 180,E1 -20258.142,E2 -20258.142} C_VEL
LIN {X 0,Y 219.941,Z 581.558,A -85,B 0,C 180,E1 -20261.051,E2 -20261.051} C_VEL
LIN {X 0,Y 220.371,Z 575.353,A -85,B 0,C 180,E1 -20264.307,E2 -20264.307} C_VEL
LIN {X 0,Y 221.354,Z 568.302,A -85,B 0,C 180,E1 -20267.17,E2 -20267.17} C_VEL
LIN {X 0,Y 222.77,Z 560.149,A -85,B 0,C 180,E1 -20269.822,E2 -20269.822} C_VEL
LIN {X 0,Y 224.493,Z 551.599,A -85,B 0,C 180,E1 -20272.064,E2 -20272.064} C_VEL
LIN {X 0,Y 226.285,Z 542.221,A -85,B 0,C 180,E1 -20274.054,E2 -20274.054} C_VEL
LIN {X 0,Y 227.072,Z 536.024,A -85,B 0,C 180,E1 -20275.184,E2 -20275.184} C_VEL
LIN {X 0,Y 226.89,Z 523.805,A -85,B 0,C 180,E1 -20277.201,E2 -20277.201} C_VEL
LIN {X 0,Y 226.455,Z 511.03,A -85,B 0,C 180,E1 -20278.878,E2 -20278.878} C_VEL
LIN {X 0,Y 225.79,Z 497.064,A -85,B 0,C 180,E1 -20280.286,E2 -20280.286} C_VEL
LIN {X 0,Y 224.881,Z 483.258,A -85,B 0,C 180,E1 -20281.26,E2 -20281.26} C_VEL
LIN {X 0,Y 223.594,Z 470.523,A -85,B 0,C 180,E1 -20281.934,E2 -20281.934} C_VEL
LIN {X 0,Y 223.214,Z 468.49,A -85,B 0,C 180,E1 -20282.098,E2 -20282.098} C_VEL
LIN {X 0,Y 222.58,Z 458.12,A -85,B 0,C 180,E1 -20283.676,E2 -20283.676} C_VEL
LIN {X 0,Y 224.278,Z 449.964,A -85,B 0,C 180,E1 -20288.427,E2 -20288.427} C_VEL
LIN {X 0,Y 225.438,Z 444.592,A -85,B 0,C 180,E1 -20291.566,E2 -20291.566} C_VEL
LIN {X 0,Y 224.738,Z 440.576,A -85,B 0,C 180,E1 -20294.007,E2 -20294.007} C_VEL
LIN {X 0,Y 223.139,Z 433.294,A -85,B 0,C 180,E1 -20298.592,E2 -20298.592} C_VEL
LIN {X 0,Y 221.838,Z 426.596,A -85,B 0,C 180,E1 -20302.992,E2 -20302.992} C_VEL
LIN {X 0,Y 220.86,Z 421.597,A -85,B 0,C 180,E1 -20306.486,E2 -20306.486} C_VEL
LIN {X 0,Y 220.86,Z 421.597,A -85,B 0,C 180,E1 -20309.394,E2 -20309.394} C_VEL
LIN {X 0,Y 220.887,Z 421.594,A -85,B 0,C 180,E1 -20313.549,E2 -20313.549} C_VEL
LIN {X 0,Y 220.869,Z 421.598,A -85,B 0,C 180,E1 -20317.553,E2 -20317.553} C_VEL
LIN {X 0,Y 220.975,Z 421.585,A -85,B 0,C 180,E1 -20322.571,E2 -20322.571} C_VEL
LIN {X 0,Y 221.017,Z 421.581,A -85,B 0,C 180,E1 -20327.139,E2 -20327.139} C_VEL
LIN {X 0,Y 221.227,Z 421.547,A -85,B 0,C 180,E1 -20330.861,E2 -20330.861} C_VEL
LIN {X 0,Y 221.281,Z 421.547,A -85,B 0,C 180,E1 -20332.702,E2 -20332.702} C_VEL
LIN {X 0,Y 221.506,Z 421.518,A -85,B 0,C 180,E1 -20338.182,E2 -20338.182} C_VEL
LIN {X 0,Y 221.507,Z 421.515,A -85,B 0,C 180,E1 -20341.819,E2 -20341.819} C_VEL
LIN {X 0,Y 221.282,Z 421.525,A -85,B 0,C 180,E1 -20347.299,E2 -20347.299} C_VEL
LIN {X 0,Y 221.104,Z 421.549,A -85,B 0,C 180,E1 -20350.995,E2 -20350.995} C_VEL
LIN {X 0,Y 221.008,Z 421.575,A -85,B 0,C 180,E1 -20356.631,E2 -20356.631} C_VEL
LIN {X 0,Y 220.885,Z 421.596,A -85,B 0,C 180,E1 -20360.487,E2 -20360.487} C_VEL
LIN {X 0,Y 220.86,Z 421.598,A -85,B 0,C 180,E1 -20364.436,E2 -20364.436} C_VEL
LIN {X 0,Y 220.82,Z 421.578,A -85,B 0,C 180,E1 -20368.517,E2 -20368.517} C_VEL
LIN {X 0,Y 220.81,Z 421.598,A -85,B 0,C 180,E1 -20372.758,E2 -20372.758} C_VEL
LIN {X 0,Y 220.804,Z 421.586,A -85,B 0,C 180,E1 -20377.28,E2 -20377.28} C_VEL
LIN {X 0,Y 220.766,Z 421.61,A -85,B 0,C 180,E1 -20381.954,E2 -20381.954} C_VEL
LIN {X 0,Y 220.829,Z 421.597,A -85,B 0,C 180,E1 -20387.054,E2 -20387.054} C_VEL
LIN {X 0,Y 220.809,Z 421.594,A -85,B 0,C 180,E1 -20390.467,E2 -20390.467} C_VEL
LIN {X 0,Y 220.832,Z 421.602,A -85,B 0,C 180,E1 -20392.797,E2 -20392.797} C_VEL
LIN {X 0,Y 220.823,Z 421.603,A -85,B 0,C 180,E1 -20397.248,E2 -20397.248} C_VEL
LIN {X 0,Y 220.879,Z 421.632,A -85,B 0,C 180,E1 -20400.706,E2 -20400.706} C_VEL
LIN {X 0,Y 221.928,Z 424.526,A -85,B 0,C 180,E1 -20400.987,E2 -20400.987} C_VEL
LIN {X 0,Y 227.636,Z 435.342,A -85,B 0,C 180,E1 -20402.47,E2 -20402.47} C_VEL
LIN {X 0,Y 231.408,Z 444.177,A -85,B 0,C 180,E1 -20403.745,E2 -20403.745} C_VEL
LIN {X 0,Y 235.108,Z 454.736,A -85,B 0,C 180,E1 -20405.396,E2 -20405.396} C_VEL
LIN {X 0,Y 236.406,Z 459.103,A -85,B 0,C 180,E1 -20406.133,E2 -20406.133} C_VEL
LIN {X 0,Y 234.873,Z 469.92,A -85,B 0,C 180,E1 -20407.575,E2 -20407.575} C_VEL
LIN {X 0,Y 232.851,Z 480.826,A -85,B 0,C 180,E1 -20409.404,E2 -20409.404} C_VEL
LIN {X 0,Y 230.928,Z 490.133,A -85,B 0,C 180,E1 -20411.366,E2 -20411.366} C_VEL
LIN {X 0,Y 228.887,Z 498.398,A -85,B 0,C 180,E1 -20413.502,E2 -20413.502} C_VEL
LIN {X 0,Y 226.893,Z 506.386,A -85,B 0,C 180,E1 -20416.112,E2 -20416.112} C_VEL
LIN {X 0,Y 225.433,Z 511.858,A -85,B 0,C 180,E1 -20418.311,E2 -20418.311} C_VEL
LIN {X 0,Y 224.103,Z 517.166,A -85,B 0,C 180,E1 -20420.981,E2 -20420.981} C_VEL
LIN {X 0,Y 222.898,Z 521.342,A -85,B 0,C 180,E1 -20423.666,E2 -20423.666} C_VEL
LIN {X 0,Y 221.992,Z 524.481,A -85,B 0,C 180,E1 -20426.372,E2 -20426.372} C_VEL
LIN {X 0,Y 221.508,Z 527.182,A -85,B 0,C 180,E1 -20430.002,E2 -20430.002} C_VEL
LIN {X 0,Y 221.505,Z 527.901,A -85,B 0,C 180,E1 -20431.82,E2 -20431.82} C_VEL
LIN {X 0,Y 221.408,Z 528.283,A -85,B 0,C 180,E1 -20435.466,E2 -20435.466} C_VEL
LIN {X 0,Y 221.823,Z 527.866,A -85,B 0,C 180,E1 -20437.283,E2 -20437.283} C_VEL
LIN {X 0,Y 223.242,Z 525.775,A -85,B 0,C 180,E1 -20440.89,E2 -20440.89} C_VEL
LIN {X 0,Y 224.599,Z 522.653,A -85,B 0,C 180,E1 -20444.06,E2 -20444.06} C_VEL
LIN {X 0,Y 226.357,Z 518.162,A -85,B 0,C 180,E1 -20447.157,E2 -20447.157} C_VEL
LIN {X 0,Y 228.15,Z 513.059,A -85,B 0,C 180,E1 -20449.808,E2 -20449.808} C_VEL
LIN {X 0,Y 230.255,Z 506.626,A -85,B 0,C 180,E1 -20452.431,E2 -20452.431} C_VEL
LIN {X 0,Y 232.859,Z 498.565,A -85,B 0,C 180,E1 -20454.997,E2 -20454.997} C_VEL
LIN {X 0,Y 235.272,Z 490.212,A -85,B 0,C 180,E1 -20457.102,E2 -20457.102} C_VEL
LIN {X 0,Y 237.774,Z 479.927,A -85,B 0,C 180,E1 -20459.191,E2 -20459.191} C_VEL
LIN {X 0,Y 239.959,Z 468.885,A -85,B 0,C 180,E1 -20460.971,E2 -20460.971} C_VEL
LIN {X 0,Y 240.403,Z 464.974,A -85,B 0,C 180,E1 -20461.54,E2 -20461.54} C_VEL
LIN {X 0,Y 237.273,Z 454.817,A -85,B 0,C 180,E1 -20463.483,E2 -20463.483} C_VEL
LIN {X 0,Y 232.335,Z 443.047,A -85,B 0,C 180,E1 -20465.613,E2 -20465.613} C_VEL
LIN {X 0,Y 227.231,Z 433.057,A -85,B 0,C 180,E1 -20467.336,E2 -20467.336} C_VEL
LIN {X 0,Y 222.64,Z 425.468,A -85,B 0,C 180,E1 -20468.642,E2 -20468.642} C_VEL
LIN {X 0,Y 221.139,Z 422.9,A -85,B 0,C 180,E1 -20469.053,E2 -20469.053} C_VEL
LIN {X 0,Y 220.991,Z 422.466,A -85,B 0,C 180,E1 -20469.154,E2 -20469.154} C_VEL
LIN {X 0,Y 220.818,Z 421.589,A -85,B 0,C 180,E1 -20469.698,E2 -20469.698} C_VEL
LIN {X 0,Y 220.777,Z 421.607,A -85,B 0,C 180,E1 -20474.455,E2 -20474.455} C_VEL
LIN {X 0,Y 220.773,Z 421.606,A -85,B 0,C 180,E1 -20478.047,E2 -20478.047} C_VEL
LIN {X 0,Y 220.812,Z 421.563,A -85,B 0,C 180,E1 -20480.464,E2 -20480.464} C_VEL
LIN {X 0,Y 220.808,Z 421.606,A -85,B 0,C 180,E1 -20485.046,E2 -20485.046} C_VEL
LIN {X 0,Y 220.84,Z 421.544,A -85,B 0,C 180,E1 -20489.39,E2 -20489.39} C_VEL
LIN {X 0,Y 220.91,Z 421.553,A -85,B 0,C 180,E1 -20492.637,E2 -20492.637} C_VEL
LIN {X 0,Y 224.733,Z 436.002,A -85,B 0,C 180,E1 -20494.597,E2 -20494.597} C_VEL
LIN {X 0,Y 228.512,Z 450.101,A -85,B 0,C 180,E1 -20496.86,E2 -20496.86} C_VEL
LIN {X 0,Y 228.919,Z 452.329,A -85,B 0,C 180,E1 -20497.233,E2 -20497.233} C_VEL
LIN {X 0,Y 227.19,Z 464.935,A -85,B 0,C 180,E1 -20499.397,E2 -20499.397} C_VEL
LIN {X 0,Y 225.405,Z 476.728,A -85,B 0,C 180,E1 -20501.832,E2 -20501.832} C_VEL
LIN {X 0,Y 224.034,Z 487.659,A -85,B 0,C 180,E1 -20504.535,E2 -20504.535} C_VEL
LIN {X 0,Y 222.832,Z 496.913,A -85,B 0,C 180,E1 -20507.245,E2 -20507.245} C_VEL
LIN {X 0,Y 221.901,Z 506.013,A -85,B 0,C 180,E1 -20510.428,E2 -20510.428} C_VEL
LIN {X 0,Y 221.16,Z 513.572,A -85,B 0,C 180,E1 -20513.614,E2 -20513.614} C_VEL
LIN {X 0,Y 220.867,Z 518.963,A -85,B 0,C 180,E1 -20516.351,E2 -20516.351} C_VEL
LIN {X 0,Y 221.163,Z 523.505,A -85,B 0,C 180,E1 -20519.089,E2 -20519.089} C_VEL
LIN {X 0,Y 221.62,Z 528.323,A -85,B 0,C 180,E1 -20522.726,E2 -20522.726} C_VEL
LIN {X 0,Y 222.451,Z 531.105,A -85,B 0,C 180,E1 -20525.438,E2 -20525.438} C_VEL
LIN {X 0,Y 224.092,Z 533.709,A -85,B 0,C 180,E1 -20529.021,E2 -20529.021} C_VEL
LIN {X 0,Y 226.592,Z 535.08,A -85,B 0,C 180,E1 -20532.539,E2 -20532.539} C_VEL
LIN {X 0,Y 229.79,Z 535.282,A -85,B 0,C 180,E1 -20535.977,E2 -20535.977} C_VEL
LIN {X 0,Y 233.596,Z 534.382,A -85,B 0,C 180,E1 -20539.326,E2 -20539.326} C_VEL
LIN {X 0,Y 238.246,Z 532.322,A -85,B 0,C 180,E1 -20542.549,E2 -20542.549} C_VEL
LIN {X 0,Y 243.64,Z 529.103,A -85,B 0,C 180,E1 -20545.638,E2 -20545.638} C_VEL
LIN {X 0,Y 249.809,Z 524.671,A -85,B 0,C 180,E1 -20548.572,E2 -20548.572} C_VEL
LIN {X 0,Y 256.636,Z 518.983,A -85,B 0,C 180,E1 -20551.353,E2 -20551.353} C_VEL
LIN {X 0,Y 264.075,Z 511.991,A -85,B 0,C 180,E1 -20553.979,E2 -20553.979} C_VEL
LIN {X 0,Y 270.083,Z 505.742,A -85,B 0,C 180,E1 -20555.838,E2 -20555.838} C_VEL
LIN {X 0,Y 270.523,Z 505.093,A -85,B 0,C 180,E1 -20556.353,E2 -20556.353} C_VEL
LIN {X 0,Y 269.928,Z 505.158,A -85,B 0,C 180,E1 -20558.673,E2 -20558.673} C_VEL
LIN {X 0,Y 269.121,Z 506.43,A -85,B 0,C 180,E1 -20561.03,E2 -20561.03} C_VEL
LIN {X 0,Y 268.847,Z 507.132,A -85,B 0,C 180,E1 -20561.885,E2 -20561.885} C_VEL
LIN {X 0,Y 267.954,Z 508.824,A -85,B 0,C 180,E1 -20562.995,E2 -20562.995} C_VEL
LIN {X 0,Y 264.067,Z 515.594,A -85,B 0,C 180,E1 -20565.681,E2 -20565.681} C_VEL
LIN {X 0,Y 262.694,Z 518.097,A -85,B 0,C 180,E1 -20566.569,E2 -20566.569} C_VEL
LIN {X 0,Y 261.353,Z 520.32,A -85,B 0,C 180,E1 -20567.229,E2 -20567.229} C_VEL
LIN {X 0,Y 258.685,Z 524.052,A -85,B 0,C 180,E1 -20568.077,E2 -20568.077} C_VEL
LIN {X 0,Y 251.233,Z 532.944,A -85,B 0,C 180,E1 -20569.842,E2 -20569.842} C_VEL
LIN {X 0,Y 247.57,Z 537.606,A -85,B 0,C 180,E1 -20571.049,E2 -20571.049} C_VEL
LIN {X 0,Y 242.726,Z 544.268,A -85,B 0,C 180,E1 -20573.071,E2 -20573.071} C_VEL
LIN {X 0,Y 235.204,Z 554.147,A -85,B 0,C 180,E1 -20576.44,E2 -20576.44} C_VEL
LIN {X 0,Y 228.492,Z 562.076,A -85,B 0,C 180,E1 -20579.595,E2 -20579.595} C_VEL
LIN {X 0,Y 222.041,Z 570.073,A -85,B 0,C 180,E1 -20583.695,E2 -20583.695} C_VEL
LIN {X 0,Y 217.909,Z 575.419,A -85,B 0,C 180,E1 -20587.229,E2 -20587.229} C_VEL
LIN {X 0,Y 214.436,Z 580.656,A -85,B 0,C 180,E1 -20591.888,E2 -20591.888} C_VEL
LIN {X 0,Y 212.836,Z 584.21,A -85,B 0,C 180,E1 -20596.634,E2 -20596.634} C_VEL
LIN {X 0,Y 212.686,Z 586.084,A -85,B 0,C 180,E1 -20600.488,E2 -20600.488} C_VEL
LIN {X 0,Y 212.833,Z 587.828,A -85,B 0,C 180,E1 -20602.408,E2 -20602.408} C_VEL
LIN {X 0,Y 213.136,Z 589.139,A -85,B 0,C 180,E1 -20604.321,E2 -20604.321} C_VEL
LIN {X 0,Y 213.426,Z 589.983,A -85,B 0,C 180,E1 -20606.222,E2 -20606.222} C_VEL
LIN {X 0,Y 213.87,Z 590.433,A -85,B 0,C 180,E1 -20608.115,E2 -20608.115} C_VEL
LIN {X 0,Y 214.365,Z 590.474,A -85,B 0,C 180,E1 -20609.998,E2 -20609.998} C_VEL
LIN {X 0,Y 213.976,Z 589.93,A -85,B 0,C 180,E1 -20611.88,E2 -20611.88} C_VEL
LIN {X 0,Y 213.584,Z 588.934,A -85,B 0,C 180,E1 -20613.771,E2 -20613.771} C_VEL
LIN {X 0,Y 213.34,Z 587.53,A -85,B 0,C 180,E1 -20615.67,E2 -20615.67} C_VEL
LIN {X 0,Y 213.007,Z 584.96,A -85,B 0,C 180,E1 -20618.182,E2 -20618.182} C_VEL
LIN {X 0,Y 212.895,Z 580.464,A -85,B 0,C 180,E1 -20621.422,E2 -20621.422} C_VEL
LIN {X 0,Y 213.405,Z 574.228,A -85,B 0,C 180,E1 -20624.785,E2 -20624.785} C_VEL
LIN {X 0,Y 214.594,Z 566.347,A -85,B 0,C 180,E1 -20628.04,E2 -20628.04} C_VEL
LIN {X 0,Y 216.03,Z 558.982,A -85,B 0,C 180,E1 -20630.468,E2 -20630.468} C_VEL
LIN {X 0,Y 217.846,Z 550.397,A -85,B 0,C 180,E1 -20632.774,E2 -20632.774} C_VEL
LIN {X 0,Y 219.943,Z 539.78,A -85,B 0,C 180,E1 -20635.046,E2 -20635.046} C_VEL
LIN {X 0,Y 220.216,Z 533.218,A -85,B 0,C 180,E1 -20636.302,E2 -20636.302} C_VEL
LIN {X 0,Y 220.117,Z 522.512,A -85,B 0,C 180,E1 -20638.093,E2 -20638.093} C_VEL
LIN {X 0,Y 219.885,Z 510.499,A -85,B 0,C 180,E1 -20639.714,E2 -20639.714} C_VEL
LIN {X 0,Y 219.336,Z 496.58,A -85,B 0,C 180,E1 -20641.174,E2 -20641.174} C_VEL
LIN {X 0,Y 218.589,Z 483.46,A -85,B 0,C 180,E1 -20642.158,E2 -20642.158} C_VEL
LIN {X 0,Y 217.523,Z 472.177,A -85,B 0,C 180,E1 -20642.785,E2 -20642.785} C_VEL
LIN {X 0,Y 216.624,Z 467.63,A -85,B 0,C 180,E1 -20643.141,E2 -20643.141} C_VEL
LIN {X 0,Y 215.909,Z 455.985,A -85,B 0,C 180,E1 -20644.957,E2 -20644.957} C_VEL
LIN {X 0,Y 217.826,Z 447.324,A -85,B 0,C 180,E1 -20650.184,E2 -20650.184} C_VEL
LIN {X 0,Y 218.196,Z 445.725,A -85,B 0,C 180,E1 -20651.152,E2 -20651.152} C_VEL
LIN {X 0,Y 218.179,Z 443.42,A -85,B 0,C 180,E1 -20652.564,E2 -20652.564} C_VEL
LIN {X 0,Y 216.615,Z 436.426,A -85,B 0,C 180,E1 -20657.052,E2 -20657.052} C_VEL
LIN {X 0,Y 215.191,Z 429.563,A -85,B 0,C 180,E1 -20661.646,E2 -20661.646} C_VEL
LIN {X 0,Y 213.962,Z 423.262,A -85,B 0,C 180,E1 -20666.055,E2 -20666.055} C_VEL
LIN {X 0,Y 213.82,Z 422.473,A -85,B 0,C 180,E1 -20666.736,E2 -20666.736} C_VEL
LIN {X 0,Y 213.773,Z 422.476,A -85,B 0,C 180,E1 -20670.453,E2 -20670.453} C_VEL
LIN {X 0,Y 213.793,Z 422.474,A -85,B 0,C 180,E1 -20674.701,E2 -20674.701} C_VEL
LIN {X 0,Y 213.804,Z 422.474,A -85,B 0,C 180,E1 -20678.803,E2 -20678.803} C_VEL
LIN {X 0,Y 213.953,Z 422.46,A -85,B 0,C 180,E1 -20682.805,E2 -20682.805} C_VEL
